VAR_INPUT
    ESS : BOOL;
    TouchSensor01 : BOOL;
    EncoderStartPosition01 : UDINT;
    EncoderStartPosition02 : UDINT;
    TOF_Time_TSR : TIME;
    AutomaticMode : BOOL;
END_VAR

VAR_OUTPUT
    DO_MovingVerticalVSG_01 : BOOL;
END_VAR

VSG_VerticalMoveWithEncoder(
    MethodCall := MethodCall_VerticalMove,
    EmergencyStopSignal := NOT ESS,
    Direction := DirectionVertical,
    InitStateDrive_Input := FALSE,
    DI01 := TouchSensor01,
    DI02_EncoderStart01 := EncoderStartPosition01,
    DI03_EncoderTarget01 := EncoderTargetPosition01,
    DI04_EncoderStart02 := EncoderStartPosition02,
    DI05_EncoderTarget02 := EncoderTargetPosition02,
    TouchSensorRelief := TSR,
    TOF_Time_MotorControl := T#0MS,
    TOF_Time_TouchSensorRelief := TOF_Time_TSR,
    OperatingMode := AutomaticMode
);

DO_MovingVerticalVSG_01 := VSG_VerticalMoveWithEncoder.DigitalOutputControl_01;
ResetMethodCall := VSG_VerticalMoveWithEncoder.ResetMethodCall;

IF ResetMethodCall THEN
    MethodCall_VerticalMove := FALSE;
    jobRunning := FALSE;
    jobFinished := TRUE;
    state := 100;
END_IF;

{attribute 'TcRpcEnable' := '1'}
METHOD Abort : HRESULT
VAR_INPUT
    hdl : UDINT;
END_VAR
callCounterAbort := callCounterAbort + 1;

MethodCall_VerticalMove := FALSE;
DO_MovingVerticalVSG_01 := FALSE;

jobRunning := FALSE;
jobFinished := TRUE;
state := 999;

Abort := 0;
END_METHOD

{attribute 'TcRpcEnable' := '1'}
METHOD CheckState : HRESULT
VAR_INPUT
    hdl : UDINT;
END_VAR

VAR_OUTPUT
    bBusy : BOOL;
    State : UDINT;
    IsDone : BOOL;
END_VAR
callCounterCheckState := callCounterCheckState + 1;

bBusy := jobRunning;
State := state;
IsDone := jobFinished;

CheckState := 0;
END_METHOD

{attribute 'TcRpcEnable' := '1'}
METHOD Start : HRESULT
VAR_INPUT
    MethodCall : BOOL;
    MovementDirection : BOOL;
    EncoderPositionVertical_01 : UDINT;
    EncoderPositionVertical_02 : UDINT;
    TouchSensorRelief : BOOL;
END_VAR

VAR_OUTPUT
    hdl : UDINT;
END_VAR
callCounterStart := callCounterStart + 1;

IF NOT jobRunning THEN

    MethodCall_VerticalMove := MethodCall;
    DirectionVertical := MovementDirection;

    EncoderTargetPosition01 := EncoderPositionVertical_01;
    EncoderTargetPosition02 := EncoderPositionVertical_02;

    TSR := TouchSensorRelief;

    jobRunning := TRUE;
    jobFinished := FALSE;
    state := 1;

    hdl := 1;
    Start := 0;

ELSE

    hdl := 0;
    Start := 16#800700AA;

END_IF;
END_METHOD

END_FUNCTION_BLOCK

// ---- POUs/Moduls/VSG_Skills/VSG_AS_RotationMoveEncoder.TcPOU
{attribute 'OPC.UA.DA.JobMethod' := 'JobMethode_RotationMove'}
FUNCTION_BLOCK VSG_AS_RotationMoveEncoder
VAR
    MethodCall_RotationMove : BOOL := FALSE;
    ResetMethodCall : BOOL := FALSE;

    DirectionRotation : BOOL := TRUE;

    EncoderTargetPosition01 : UDINT;
    EncoderTargetPosition02 : UDINT;

    TSR : BOOL := FALSE;

    callCounterStart : ULINT;
    callCounterCheckState : ULINT;
    callCounterAbort : ULINT;

    jobRunning : BOOL := FALSE;
    jobFinished : BOOL := FALSE;
    state : UDINT := 0;

    VSG_RotationMoveWithEncoder : AxisControl_Encoder;
END_VAR

VAR_INPUT
    ESS : BOOL;
    TouchSensor01 : BOOL;
    EncoderStartPosition01 : UDINT;
    EncoderStartPosition02 : UDINT;
    TOF_Time_TSR : TIME;
    AutomaticMode : BOOL;
END_VAR

VAR_OUTPUT
    DO_MovingRotationVSG_01 : BOOL;
END_VAR

VSG_RotationMoveWithEncoder(
    MethodCall := MethodCall_RotationMove,
    EmergencyStopSignal := NOT ESS,
    Direction := DirectionRotation,
    InitStateDrive_Input := FALSE,
    DI01 := TouchSensor01,
    DI02_EncoderStart01 := EncoderStartPosition01,
    DI03_EncoderTarget01 := EncoderTargetPosition01,
    DI04_EncoderStart02 := EncoderStartPosition02,
    DI05_EncoderTarget02 := EncoderTargetPosition02,
    TouchSensorRelief := TSR,
    TOF_Time_MotorControl := T#0MS,
    TOF_Time_TouchSensorRelief := TOF_Time_TSR,
    OperatingMode := AutomaticMode
);

DO_MovingRotationVSG_01 := VSG_RotationMoveWithEncoder.DigitalOutputControl_01;
ResetMethodCall := VSG_RotationMoveWithEncoder.ResetMethodCall;

IF ResetMethodCall THEN
    MethodCall_RotationMove := FALSE;
    jobRunning := FALSE;
    jobFinished := TRUE;
    state := 100;
END_IF;

{attribute 'TcRpcEnable' := '1'}
METHOD Abort : HRESULT
VAR_INPUT
    hdl : UDINT;
END_VAR
callCounterAbort := callCounterAbort + 1;

MethodCall_RotationMove := FALSE;
DO_MovingRotationVSG_01 := FALSE;

jobRunning := FALSE;
jobFinished := TRUE;
state := 999;

Abort := 0;
END_METHOD

{attribute 'TcRpcEnable' := '1'}
METHOD CheckState : HRESULT
VAR_INPUT
    hdl : UDINT;
END_VAR

VAR_OUTPUT
    bBusy : BOOL;
    State : UDINT;
    IsDone : BOOL;
END_VAR
callCounterCheckState := callCounterCheckState + 1;

bBusy := jobRunning;
State := state;
IsDone := jobFinished;

CheckState := 0;
END_METHOD

{attribute 'TcRpcEnable' := '1'}
METHOD Start : HRESULT
VAR_INPUT
    MethodCall : BOOL;
    MovementDirection : BOOL;
    EncoderPositionRotation_01 : UDINT;
    EncoderPositionRotation_02 : UDINT;
    TouchSensorRelief : BOOL;
END_VAR

VAR_OUTPUT
    hdl : UDINT;
END_VAR
callCounterStart := callCounterStart + 1;

IF NOT jobRunning THEN

    MethodCall_RotationMove := MethodCall;
    DirectionRotation := MovementDirection;

    EncoderTargetPosition01 := EncoderPositionRotation_01;
    EncoderTargetPosition02 := EncoderPositionRotation_02;

    TSR := TouchSensorRelief;

    jobRunning := TRUE;
    jobFinished := FALSE;
    state := 1;

    hdl := 1;
    Start := 0;

ELSE

    hdl := 0;
    Start := 16#800700AA;

END_IF;
END_METHOD

END_FUNCTION_BLOCK

// ---- POUs/Moduls/VSG_Skills/VSG_AS_CompressorControl.TcPOU
{attribute 'OPC.UA.DA.JobMethod' := 'JobMethode_CompressorControl'}
FUNCTION_BLOCK VSG_AS_CompressorControl
VAR
    MethodCall_CompressorControl : BOOL := FALSE;
    ResetMethodCall : BOOL := FALSE;

    Destination : BOOL := TRUE;

    EncoderTargetPosition01 : UDINT;
    EncoderTargetPosition02 : UDINT;
    EncoderTargetPosition03 : UDINT;
    EncoderTargetPosition04 : UDINT;
    EncoderTargetPosition05 : UDINT;
    EncoderTargetPosition06 : UDINT;

    callCounterStart : ULINT;
    callCounterCheckState : ULINT;
    callCounterAbort : ULINT;

    jobRunning : BOOL := FALSE;
    jobFinished : BOOL := FALSE;
    state : UDINT := 0;

    MBS_VSG_VerticalMove : CompressorControl;

    TON_TimeCompressor : TIME := T#0MS;
    TON_TimeValve : TIME := T#0MS;
    TON_TimePowerOffSelfSet : TIME := T#100MS;

    PowerOffSelfSet : BOOL := TRUE;
END_VAR

VAR_INPUT
    ESS : BOOL;

    EncoderStartPosition01 : UDINT;
    EncoderStartPosition02 : UDINT;
    EncoderStartPosition03 : UDINT;
    EncoderStartPosition04 : UDINT;
    EncoderStartPosition05 : UDINT;
    EncoderStartPosition06 : UDINT;

    WorkpieceAtPickupPosition : BOOL;
    AutomaticMode : BOOL;
END_VAR

VAR_OUTPUT
    DO_CompressorVSG : BOOL;
    DO_ValveVSG : BOOL;

    VSG_ErrorDetected : BOOL;
    VSG_ErrorCode : UDINT;
END_VAR

//VSG_ErrorDetected := FALSE;
//VSG_ErrorCode := 0;

IF MethodCall_CompressorControl AND NOT WorkpieceAtPickupPosition THEN

    VSG_ErrorDetected := TRUE;
    VSG_ErrorCode := 1001;

    DO_CompressorVSG := FALSE;
    DO_ValveVSG := FALSE;

    MethodCall_CompressorControl := FALSE;
    ResetMethodCall := TRUE;

    jobRunning := FALSE;
    jobFinished := TRUE;
    state := 900;

ELSE

    MBS_VSG_VerticalMove(
        MethodCall := MethodCall_CompressorControl,
        EmergencyStopSignal := NOT ESS,
        Destination := Destination,
        InitStateDrive_Input := FALSE,

        DI01 := WorkpieceAtPickupPosition,
        DI02 := FALSE,

        DI03_EncoderStart01 := EncoderStartPosition01,
        DI04_EncoderStart02 := EncoderStartPosition02,
        DI05_EncoderStart03 := EncoderStartPosition03,
        DI06_EncoderStart04 := EncoderStartPosition04,
        DI07_EncoderStart05 := EncoderStartPosition05,
        DI08_EncoderStart06 := EncoderStartPosition06,

        DI09_EncoderTarget01 := EncoderTargetPosition01,
        DI10_EncoderTarget02 := EncoderTargetPosition02,
        DI11_EncoderTarget03 := EncoderTargetPosition03,
        DI12_EncoderTarget04 := EncoderTargetPosition04,
        DI13_EncoderTarget05 := EncoderTargetPosition05,
        DI14_EncoderTarget06 := EncoderTargetPosition06,

        PowerOFF_SelfSet := PowerOffSelfSet,
        TON_Time_PowerOFFSelfSet := TON_TimePowerOffSelfSet,
        TON_Time_Compressor := TON_TimeCompressor,
        TON_Time_Valve := TON_TimeValve,
        OperatingMode := AutomaticMode
    );

    DO_CompressorVSG := MBS_VSG_VerticalMove.DigitalOutputControl_01;
    DO_ValveVSG := MBS_VSG_VerticalMove.DigitalOutputControl_02;
    ResetMethodCall := MBS_VSG_VerticalMove.ResetMethodCall;

    IF ResetMethodCall THEN
        MethodCall_CompressorControl := FALSE;
        jobRunning := FALSE;
        jobFinished := TRUE;
        state := 100;
    END_IF;

END_IF;

{attribute 'TcRpcEnable' := '1'}
METHOD Abort : HRESULT
VAR_INPUT
    hdl : UDINT;
END_VAR
callCounterAbort := callCounterAbort + 1;

MethodCall_CompressorControl := FALSE;
ResetMethodCall := TRUE;

DO_CompressorVSG := FALSE;
DO_ValveVSG := FALSE;

jobRunning := FALSE;
jobFinished := TRUE;
state := 999;

Abort := 0;
END_METHOD

{attribute 'TcRpcEnable' := '1'}
METHOD CheckState : HRESULT
VAR_INPUT
    hdl : UDINT;
END_VAR

VAR_OUTPUT
    bBusy : BOOL;
    State : UDINT;
    IsDone : BOOL;
    HasError : BOOL;
    ErrorCode : UDINT;
END_VAR
callCounterCheckState := callCounterCheckState + 1;

bBusy := jobRunning;
State := state;
IsDone := jobFinished;
HasError := VSG_ErrorDetected;
ErrorCode := VSG_ErrorCode;

CheckState := 0;
END_METHOD

{attribute 'TcRpcEnable' := '1'}
METHOD Start : HRESULT
VAR_INPUT
    MethodCall : BOOL;
    DestinationReached : BOOL;
    EncoderTargetPosition_01 : UDINT;
    EncoderTargetPosition_02 : UDINT;
    EncoderTargetPosition_03 : UDINT;
    EncoderTargetPosition_04 : UDINT;
    EncoderTargetPosition_05 : UDINT;
    EncoderTargetPosition_06 : UDINT;
END_VAR

VAR_OUTPUT
    hdl : UDINT;
END_VAR
callCounterStart := callCounterStart + 1;

IF NOT jobRunning THEN
	
	IF MethodCall THEN
        OPCUA.lastExecutedProcess := 'VSG_Skill_SuctionProcess';
        OPCUA.lastExecutedSkill := 'VSG_AS_CompressorControl';
    END_IF;
	
    MethodCall_CompressorControl := MethodCall;
    Destination := DestinationReached;

    EncoderTargetPosition01 := EncoderTargetPosition_01;
    EncoderTargetPosition02 := EncoderTargetPosition_02;
    EncoderTargetPosition03 := EncoderTargetPosition_03;
    EncoderTargetPosition04 := EncoderTargetPosition_04;
    EncoderTargetPosition05 := EncoderTargetPosition_05;
    EncoderTargetPosition06 := EncoderTargetPosition_06;

    jobRunning := TRUE;
    jobFinished := FALSE;
    state := 1;

    hdl := 1;
    Start := 0;

ELSE

    hdl := 0;
    Start := 16#800700AA;

END_IF;
END_METHOD

END_FUNCTION_BLOCK

// ---- POUs/AtomicSkillsSchablonen/CompressorControl.TcPOU
FUNCTION_BLOCK CompressorControl
VAR_INPUT
    MethodCall : BOOL;
    EmergencyStopSignal : BOOL;
    Destination : BOOL;
    InitStateDrive_Input : BOOL;

    DI01 : BOOL;
    DI02 : BOOL;

    DI03_EncoderStart01 : UDINT;
    DI04_EncoderStart02 : UDINT;
    DI05_EncoderStart03 : UDINT;
    DI06_EncoderStart04 : UDINT;
    DI07_EncoderStart05 : UDINT;
    DI08_EncoderStart06 : UDINT;

    DI09_EncoderTarget01 : UDINT;
    DI10_EncoderTarget02 : UDINT;
    DI11_EncoderTarget03 : UDINT;
    DI12_EncoderTarget04 : UDINT;
    DI13_EncoderTarget05 : UDINT;
    DI14_EncoderTarget06 : UDINT;

    PowerOFF_SelfSet : BOOL;
    TON_Time_PowerOFFSelfSet : TIME;
    TON_Time_Compressor : TIME;
    TON_Time_Valve : TIME;
    OperatingMode : BOOL;
END_VAR

VAR_OUTPUT
    DigitalOutputControl_01 : BOOL;
    DigitalOutputControl_02 : BOOL;
    ResetMethodCall : BOOL;
END_VAR

VAR
    RS_Compressor : RS;
    RS_Valve : RS;

    TON_Compressor_Control : TON;
    TON_Valve_Control : TON;
    TON_SelfSet : TON;

    R_TRIG_MethodCall : R_TRIG;

    R_TRIG_EncoderPos01_CompressorInput : R_TRIG;
    R_TRIG_EncoderPos02_CompressorInput : R_TRIG;
    R_TRIG_EncoderPos03_CompressorInput : R_TRIG;
    R_TRIG_EncoderPos04_CompressorInput : R_TRIG;
    R_TRIG_EncoderPos05_CompressorInput : R_TRIG;
    R_TRIG_EncoderPos06_CompressorInput : R_TRIG;

    R_TRIG_EncoderPos01_CompressorOutput : R_TRIG;
    R_TRIG_EncoderPos02_CompressorOutput : R_TRIG;
    R_TRIG_EncoderPos03_CompressorOutput : R_TRIG;
    R_TRIG_EncoderPos04_CompressorOutput : R_TRIG;
    R_TRIG_EncoderPos05_CompressorOutput : R_TRIG;
    R_TRIG_EncoderPos06_CompressorOutput : R_TRIG;

    R_TRIG_EncoderPos01_ValveInput : R_TRIG;
    R_TRIG_EncoderPos02_ValveInput : R_TRIG;
    R_TRIG_EncoderPos03_ValveInput : R_TRIG;
    R_TRIG_EncoderPos04_ValveInput : R_TRIG;
    R_TRIG_EncoderPos05_ValveInput : R_TRIG;
    R_TRIG_EncoderPos06_ValveInput : R_TRIG;

    R_TRIG_EncoderPos01_ValveOutput : R_TRIG;
    R_TRIG_EncoderPos02_ValveOutput : R_TRIG;
    R_TRIG_EncoderPos03_ValveOutput : R_TRIG;
    R_TRIG_EncoderPos04_ValveOutput : R_TRIG;
    R_TRIG_EncoderPos05_ValveOutput : R_TRIG;
    R_TRIG_EncoderPos06_ValveOutput : R_TRIG;

    bEncoderInputCondition : BOOL;
    bEncoderOutputCondition : BOOL;
    bStartCondition : BOOL;
    bResetCondition : BOOL;
END_VAR

R_TRIG_MethodCall(CLK := MethodCall);

R_TRIG_EncoderPos01_CompressorInput(CLK := DI03_EncoderStart01 <> DI09_EncoderTarget01);
R_TRIG_EncoderPos02_CompressorInput(CLK := DI04_EncoderStart02 <> DI10_EncoderTarget02);
R_TRIG_EncoderPos03_CompressorInput(CLK := DI05_EncoderStart03 <> DI11_EncoderTarget03);
R_TRIG_EncoderPos04_CompressorInput(CLK := DI06_EncoderStart04 <> DI12_EncoderTarget04);
R_TRIG_EncoderPos05_CompressorInput(CLK := DI07_EncoderStart05 <> DI13_EncoderTarget05);
R_TRIG_EncoderPos06_CompressorInput(CLK := DI08_EncoderStart06 <> DI14_EncoderTarget06);

R_TRIG_EncoderPos01_CompressorOutput(CLK := DI03_EncoderStart01 = DI09_EncoderTarget01);
R_TRIG_EncoderPos02_CompressorOutput(CLK := DI04_EncoderStart02 = DI10_EncoderTarget02);
R_TRIG_EncoderPos03_CompressorOutput(CLK := DI05_EncoderStart03 = DI11_EncoderTarget03);
R_TRIG_EncoderPos04_CompressorOutput(CLK := DI06_EncoderStart04 = DI12_EncoderTarget04);
R_TRIG_EncoderPos05_CompressorOutput(CLK := DI07_EncoderStart05 = DI13_EncoderTarget05);
R_TRIG_EncoderPos06_CompressorOutput(CLK := DI08_EncoderStart06 = DI14_EncoderTarget06);

R_TRIG_EncoderPos01_ValveInput(CLK := DI03_EncoderStart01 <> DI09_EncoderTarget01);
R_TRIG_EncoderPos02_ValveInput(CLK := DI04_EncoderStart02 <> DI10_EncoderTarget02);
R_TRIG_EncoderPos03_ValveInput(CLK := DI05_EncoderStart03 <> DI11_EncoderTarget03);
R_TRIG_EncoderPos04_ValveInput(CLK := DI06_EncoderStart04 <> DI12_EncoderTarget04);
R_TRIG_EncoderPos05_ValveInput(CLK := DI07_EncoderStart05 <> DI13_EncoderTarget05);
R_TRIG_EncoderPos06_ValveInput(CLK := DI08_EncoderStart06 <> DI14_EncoderTarget06);

R_TRIG_EncoderPos01_ValveOutput(CLK := DI03_EncoderStart01 = DI09_EncoderTarget01);
R_TRIG_EncoderPos02_ValveOutput(CLK := DI04_EncoderStart02 = DI10_EncoderTarget02);
R_TRIG_EncoderPos03_ValveOutput(CLK := DI05_EncoderStart03 = DI11_EncoderTarget03);
R_TRIG_EncoderPos04_ValveOutput(CLK := DI06_EncoderStart04 = DI12_EncoderTarget04);
R_TRIG_EncoderPos05_ValveOutput(CLK := DI07_EncoderStart05 = DI13_EncoderTarget05);
R_TRIG_EncoderPos06_ValveOutput(CLK := DI08_EncoderStart06 = DI14_EncoderTarget06);

bEncoderInputCondition :=
    R_TRIG_EncoderPos01_CompressorInput.Q
    AND R_TRIG_EncoderPos02_CompressorInput.Q
    AND R_TRIG_EncoderPos03_CompressorInput.Q
    AND R_TRIG_EncoderPos04_CompressorInput.Q
    AND R_TRIG_EncoderPos05_CompressorInput.Q
    AND R_TRIG_EncoderPos06_CompressorInput.Q;

bEncoderOutputCondition :=
    R_TRIG_EncoderPos01_CompressorOutput.Q
    AND R_TRIG_EncoderPos02_CompressorOutput.Q
    AND R_TRIG_EncoderPos03_CompressorOutput.Q
    AND R_TRIG_EncoderPos04_CompressorOutput.Q
    AND R_TRIG_EncoderPos05_CompressorOutput.Q
    AND R_TRIG_EncoderPos06_CompressorOutput.Q;

bStartCondition :=
    (DI01 OR bEncoderInputCondition OR InitStateDrive_Input)
    AND OperatingMode;

bResetCondition :=
    (Destination AND (DI02 OR bEncoderOutputCondition))
    OR EmergencyStopSignal;

ResetMethodCall := bResetCondition;

RS_Compressor(
    SET := R_TRIG_MethodCall.Q AND bStartCondition,
    RESET1 := bResetCondition
);

TON_Compressor_Control(
    IN := RS_Compressor.Q1,
    PT := TON_Time_Compressor
);

DigitalOutputControl_01 := TON_Compressor_Control.Q;

TON_SelfSet(
    IN := R_TRIG_MethodCall.Q AND PowerOFF_SelfSet,
    PT := TON_Time_PowerOFFSelfSet
);

RS_Valve(
    SET := R_TRIG_MethodCall.Q AND (DI01 OR bEncoderInputCondition OR InitStateDrive_Input),
    RESET1 := (Destination AND (DI02 OR bEncoderOutputCondition OR TON_SelfSet.Q)) OR EmergencyStopSignal
);

TON_Valve_Control(
    IN := RS_Valve.Q1,
    PT := TON_Time_Valve
);

DigitalOutputControl_02 := TON_Valve_Control.Q;

END_FUNCTION_BLOCK

// ---- POUs/ControlOfOutputs/VSG_ControlOfOutputs.TcPOU
FUNCTION_BLOCK VSG_ControlOfOutputs
VAR_INPUT
	F4							: BOOL;
	F1							: BOOL;
	A2							: BOOL;
	A1							: BOOL;
	A6							: BOOL;
	Start						: BOOL;
	VSG_VertikalDown01			: BOOL; 
	VSG_VertikalDown02			: BOOL; 
	VSG_VertikalUp01			: BOOL;
	VSG_VertikalUp02			: BOOL; 
	VSG_HorizontalForwards01 	: BOOL; 
	VSG_HorizontalForwards02	: BOOL;
	VSG_HorizontalBackwards01 	: BOOL; 
	VSG_HorizontalBackwards02 	: BOOL;
	VSG_RotationCW01		 	: BOOL; 
	VSG_RotationCW02		 	: BOOL;
	VSG_RotationCCW01		 	: BOOL; 
	VSG_RotationCCW02		 	: BOOL;
	VSG_Compressor				: BOOL;
	VSG_Valve					: BOOL;
	Init_VSG_VertikalUp			: BOOL;
	Init_VSG_VertikalDown		: BOOL;	
	Init_VSG_HorizontalForwards : BOOL;
	Init_VSG_HorizontalBackwards: BOOL;
	Init_VSG_RotationCW			: BOOL;
	Init_VSG_RotationCCW		: BOOL;

END_VAR
VAR_OUTPUT
	MoveVerticalDown : BOOL;
	MoveVerticalUp : BOOL;
	MoveHorizontalForwards : BOOL;
	MoveHorizontalBackwards : BOOL;
	MoveRotationCW	: BOOL;
	MoveRotationCCW : BOOL;
	CompressorON : BOOL;
	ValveON : BOOL;
	Light_Q1: BOOL;
	Light_Q2: BOOL;
	Light_Q3: BOOL;
END_VAR
VAR
END_VAR

MoveVerticalDown := ((((((F1) OR (A2))) AND (((VSG_VertikalDown01) OR (VSG_VertikalDown02) OR (Init_VSG_VertikalDown))))) OR (((Start) AND (F4))));
MoveVerticalUp := ((((((F1) OR (A2))) AND (((VSG_VertikalUp01) OR (VSG_VertikalUp02) OR (Init_VSG_VertikalUp))))) OR (((Start) AND (F4))));
MoveHorizontalForwards := ((((((F1) OR (A2))) AND (((VSG_HorizontalForwards01) OR (VSG_HorizontalForwards02) OR (Init_VSG_HorizontalForwards))))) OR (((Start) AND (F4))));
MoveHorizontalBackwards := ((((((F1) OR (A2))) AND (((VSG_HorizontalBackwards01) OR (VSG_HorizontalBackwards02) OR (Init_VSG_HorizontalBackwards))))) OR (((Start) AND (F4))));
MoveRotationCW := ((((((F1) OR (A2))) AND (((VSG_RotationCW01) OR (VSG_RotationCW02) OR (Init_VSG_RotationCW))))) OR (((Start) AND (F4))));
MoveRotationCCW := ((((((F1) OR (A2))) AND (((VSG_RotationCCW01) OR (VSG_RotationCCW02) OR (Init_VSG_RotationCCW))))) OR (((Start) AND (F4))));
CompressorON := ((((((F1) OR (A2))) AND (VSG_Compressor))) OR (((Start) AND (F4))));
ValveON := ((((((F1) OR (A2))) AND (VSG_Valve))) OR (((Start) AND (F4))));
Light_Q1 := F1;
Light_Q2 := F4;
Light_Q3 := A1;

END_FUNCTION_BLOCK

// ---- POUs/OperatingModes/VSG_OperatingModes.TcPOU
FUNCTION_BLOCK VSG_OperatingModes
VAR_INPUT
	Start 			: BOOL;
	Stop			: BOOL;
	Reset			: BOOL;
	Schalter		: BOOL;
	Schrittkette_GS	: BOOL;
	Count1 : INT := 0;
	Count2 : INT := 0;
	Alt_abort: BOOL;
	Err_detected: BOOL;
	Diag_finished: BOOL;
	Alt_found: BOOL;
	Cycle_finished: BOOL;

END_VAR
VAR_OUTPUT
	{attribute 'OPC.UA.DA' := '1'} // für OPC UA freigeben
	A1 : BOOL := FALSE; //Initialzustand
	{attribute 'OPC.UA.DA' := '1'} // für OPC UA freigeben
	A2 : BOOL; //Stillstand angefordert am Ende des Zyklus
//	A3 : BOOL; //Stillstand angefordert in einem bestimmten Zustand
//	A4 : BOOL; //Erhaltener Stillstand
	{attribute 'OPC.UA.DA' := '1'} // für OPC UA freigeben
	A5 : BOOL; //Vorbereitung zur Wiederaufnahme nach Störung
	{attribute 'OPC.UA.DA' := '1'} // für OPC UA freigeben
	A6 : BOOL; //Fahrt in den Initialzustand
	{attribute 'OPC.UA.DA' := '1'} // für OPC UA freigeben
	F1 : BOOL; //Normalbetrieb
//	F2 : BOOL; //Anfahren
//	F3 : BOOL; //Abfahren
	{attribute 'OPC.UA.DA' := '1'} // für OPC UA freigeben
	F4 : BOOL; //Handbetrieb
//	F5 : BOOL; //Schrittbetrieb
//	F6 : BOOL; //Testbetrieb
{attribute 'OPC.UA.DA' := '1'} // für OPC UA freigeben
	D1 : BOOL; //Not-Aus
	{attribute 'OPC.UA.DA' := '1'} // für OPC UA freigeben
	D2 : BOOL; //Diagnose und Störbehandlung
	{attribute 'OPC.UA.DA' := '1'} // für OPC UA freigeben
	D3 : BOOL; //Produktion trotz Störung
	MethodCall_InitStateDrive : BOOL;
	InputVar_InitStateDrive : BOOL;
END_VAR
VAR
	bFirstScan : BOOL := TRUE;
	FirstScanCount: INT := 0;
	AlwaysTrue : BOOL := TRUE;
	TestingVariable : BOOL;	
	 nTaskIdx : DINT;
	RS_InitialState: RS;
	RS_InitialState11: RS;	
	RS_InitialDrive: RS;
	RS_ManualOperationMode: RS;
	RS_AutomaticOperationMode: RS;
	RS_CycleEnded: RS;
	//Count: INT := 0;
	R_TRIG_Manual: R_TRIG;
	R_TRIG_Automatic: R_TRIG;
	R_TRIG_InitialDrive: R_TRIG;
	R_TRIG_CycleEnded: R_TRIG;
	R_TRIG_Init: R_TRIG;
	NeverTrue: BOOL := FALSE;
	SR_D1: SR;
	RS_D2: RS;
	
	RS_D3: RS;
	RS_A5: RS;
	
	
	bFirstCycle: BOOL;
END_VAR
VAR // added by the converter: edge detectors and wires of the graphical bodies
    _w1, _w2, _w3, _w4 : BOOL;
END_VAR

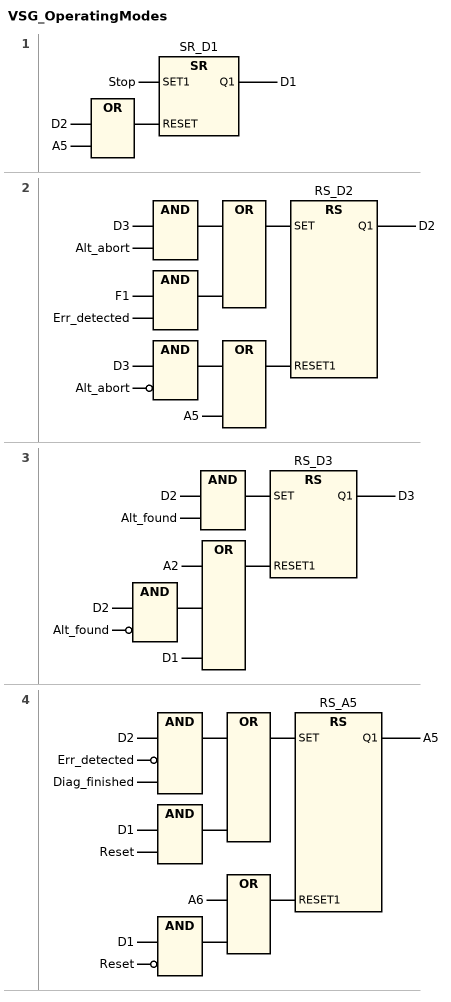
// NETWORK 1
SR_D1(SET1 := Stop, RESET := D2 OR A5); // SR
D1 := SR_D1.Q1;

// NETWORK 2
RS_D2(SET := D3 AND Alt_abort OR F1 AND Err_detected, RESET1 := D3 AND NOT Alt_abort OR A5); // RS
D2 := RS_D2.Q1;

// NETWORK 3
RS_D3(SET := D2 AND Alt_found, RESET1 := A2 OR D2 AND NOT Alt_found OR D1); // RS
D3 := RS_D3.Q1;

// NETWORK 4
RS_A5(SET := D2 AND NOT Err_detected AND Diag_finished OR D1 AND Reset, RESET1 := A6 OR D1 AND NOT Reset); // RS
A5 := RS_A5.Q1;

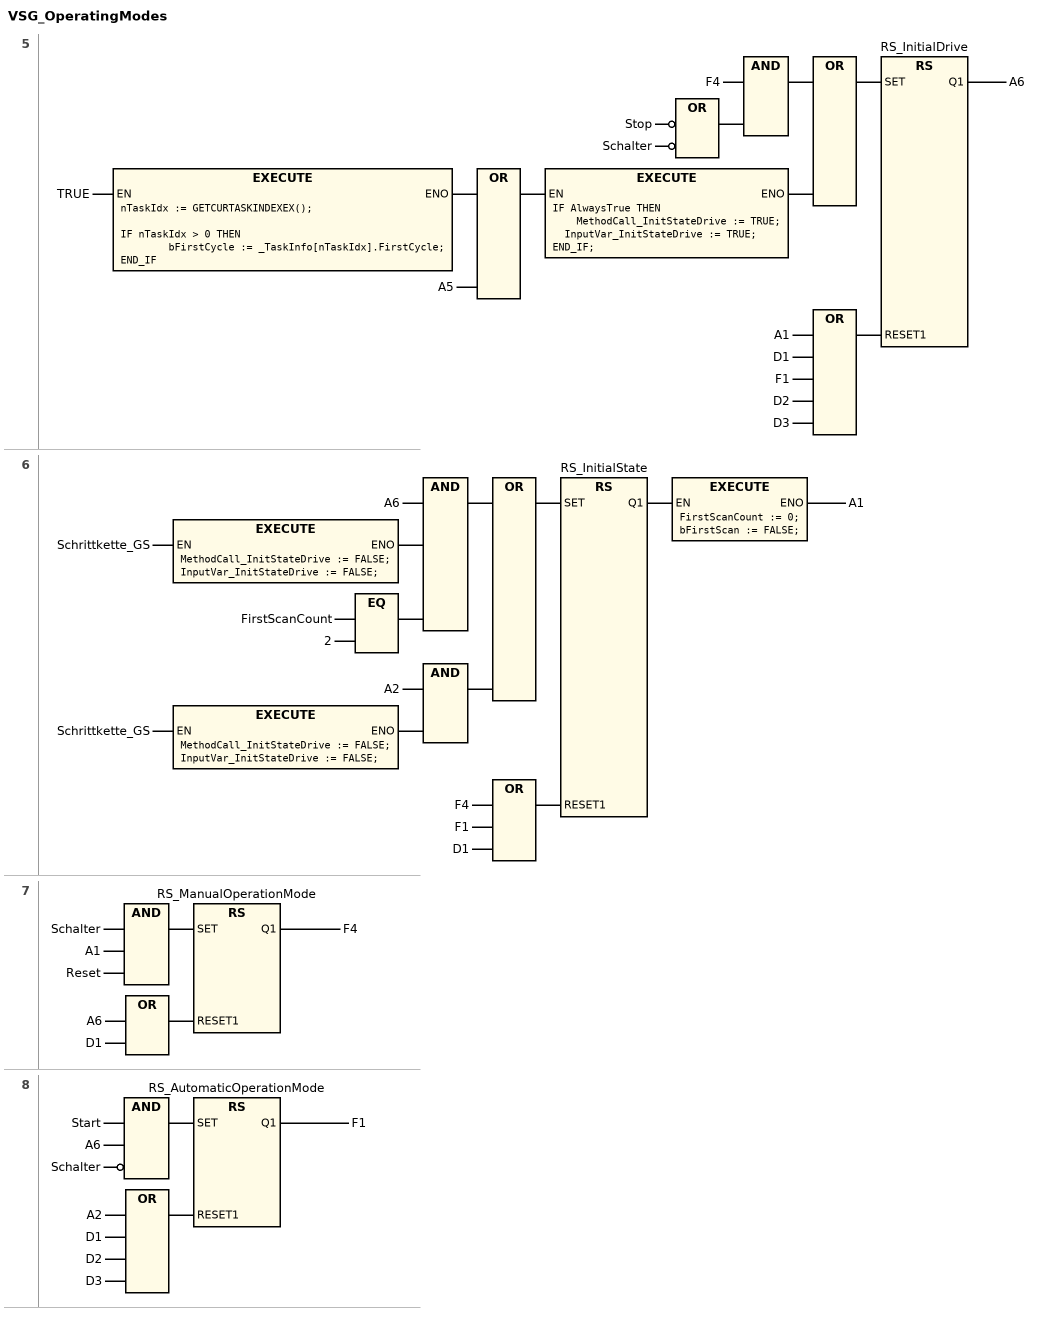
// NETWORK 5
nTaskIdx := GETCURTASKINDEXEX();

IF nTaskIdx > 0 THEN
        bFirstCycle := _TaskInfo[nTaskIdx].FirstCycle;
END_IF
_w1 := TRUE OR A5;
IF _w1 THEN
    IF AlwaysTrue THEN
        MethodCall_InitStateDrive := TRUE;
    	InputVar_InitStateDrive := TRUE;
    END_IF;
END_IF
RS_InitialDrive(SET := F4 AND (NOT Stop OR NOT Schalter) OR _w1, RESET1 := A1 OR D1 OR F1 OR D2 OR D3); // RS
A6 := RS_InitialDrive.Q1;

// NETWORK 6
_w2 := Schrittkette_GS;
IF _w2 THEN
    MethodCall_InitStateDrive := FALSE;
    InputVar_InitStateDrive := FALSE;
END_IF
_w3 := Schrittkette_GS;
IF _w3 THEN
    MethodCall_InitStateDrive := FALSE;
    InputVar_InitStateDrive := FALSE;
END_IF
RS_InitialState(SET := A6 AND _w2 AND FirstScanCount = 2 OR A2 AND _w3, RESET1 := F4 OR F1 OR D1); // RS
_w4 := RS_InitialState.Q1;
IF _w4 THEN
    FirstScanCount := 0;
    bFirstScan := FALSE;
END_IF
A1 := _w4;

// NETWORK 7
RS_ManualOperationMode(SET := Schalter AND A1 AND Reset, RESET1 := A6 OR D1); // RS
F4 := RS_ManualOperationMode.Q1;

// NETWORK 8
RS_AutomaticOperationMode(SET := Start AND A6 AND NOT Schalter, RESET1 := A2 OR D1 OR D2 OR D3); // RS
F1 := RS_AutomaticOperationMode.Q1;

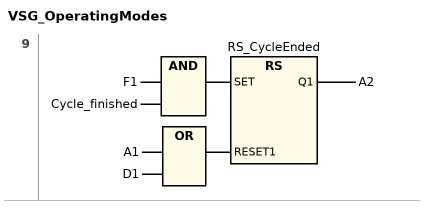
// NETWORK 9
RS_CycleEnded(SET := F1 AND Cycle_finished, RESET1 := A1 OR D1); // RS
A2 := RS_CycleEnded.Q1;

END_FUNCTION_BLOCK

// ---- POUs/DiagnosisHandler/VSG_DiagnosisHandler.TcPOU
FUNCTION_BLOCK VSG_DiagnosisHandler
VAR_INPUT
    Diagnose_gefordert : BOOL;
    ErrorDetectedRaw   : BOOL;
    Reset              : BOOL;
    PulseTime          : TIME := T#100MS;
END_VAR
VAR_OUTPUT
    Err_detected  : BOOL := FALSE;
    Diag_finished : BOOL := FALSE;
    Alt_found     : BOOL := FALSE;
    Busy          : BOOL := FALSE;
END_VAR
VAR
    rtReq      : R_TRIG;
    rtError    : R_TRIG;
    rtDiagAck  : R_TRIG;
    rtAltFound : R_TRIG;
    tpPulse    : TP;
END_VAR

rtReq(CLK := Diagnose_gefordert);
rtError(CLK := ErrorDetectedRaw);
rtDiagAck(CLK := OPCUA.Diag_finished);
rtAltFound(CLK := OPCUA.Alt_found);

IF Reset THEN
    Err_detected := FALSE;
    Diag_finished := FALSE;
    Alt_found := FALSE;
    Busy := FALSE;
    OPCUA.TriggerD2 := FALSE;
END_IF

IF rtError.Q THEN
    Err_detected := TRUE;
    Diag_finished := FALSE;
    Alt_found := FALSE;
	OPCUA.TriggerD2 := TRUE;
END_IF

IF rtReq.Q AND Err_detected AND NOT Busy THEN
    Busy := TRUE;
END_IF

IF OPCUA.TriggerD2 AND Diag_finished THEN
    OPCUA.TriggerD2 := FALSE;
END_IF

IF Busy AND rtDiagAck.Q THEN
    Diag_finished := TRUE;
    Alt_found := FALSE;
    Busy := FALSE;
    OPCUA.Diag_finished := FALSE;
    OPCUA.TriggerD2 := FALSE;
END_IF

IF Busy AND rtAltFound.Q THEN
    Alt_found := TRUE;
    Diag_finished := TRUE;
    Busy := FALSE;
    OPCUA.Alt_found := FALSE;
    OPCUA.TriggerD2 := FALSE;
END_IF

IF NOT Diagnose_gefordert AND (Diag_finished OR Alt_found) THEN
    Err_detected := FALSE;
    Diag_finished := FALSE;
    Alt_found := FALSE;
END_IF

END_FUNCTION_BLOCK

// ---- POUs/InitStateDrive/VSG_InitialStateDrive.TcPOU
FUNCTION_BLOCK VSG_InitialStateDrive
VAR_INPUT
    MethodCall_InitDrive : BOOL;
    ESS : BOOL;
    InputInitDriveMode : BOOL;

    TouchSensor01_Rotation : BOOL;
    TouchSensor02_Vertical : BOOL;
    TouchSensor03_horizontal : BOOL;

    TOF_Time_TSR : TIME;
    InitDriveMode : BOOL;
END_VAR

VAR_OUTPUT
    VSG_Init_RotateCW : BOOL;
    VSG_Init_RotateCCW : BOOL;

    VSG_Init_VerticalUp : BOOL;
    VSG_Init_VerticalDown : BOOL;

    VSG_Init_HorizontalForwards : BOOL;
    VSG_Init_HorizontalBackwards : BOOL;

    ResetMethodCall_RotateCW : BOOL;
    ResetMethodCall_RGB_Vertical : BOOL;
    ResetMethodCall_RGB_Horizontal : BOOL;
END_VAR

VAR
    TSR : BOOL := TRUE;

    DirectionVertical : BOOL := TRUE;
    DirectionHorizontal : BOOL := TRUE;
    DirectionRotation : BOOL := TRUE;

    VSG_InitDrive_Rotate_CW : AxisControl_MultipleInputSensors;
    VSG_InitDrive_Vertical_Up : AxisControl_MultipleInputSensors;
    VSG_InitDrive_Horizontal_Backwards : AxisControl_MultipleInputSensors;
END_VAR

VSG_InitDrive_Rotate_CW(
    MethodCall := MethodCall_InitDrive,
    EmergencyStopSignal := NOT ESS,
    Direction := DirectionRotation,
    InitStateDrive_Input := InputInitDriveMode,
    DI01 := FALSE,
    DI02 := TouchSensor01_Rotation,
    TouchSensorRelief := TSR,
    TOF_Time_MotorControl := T#0MS,
    TOF_Time_TouchSensorRelief := TOF_Time_TSR,
    OperatingMode := InitDriveMode
);

VSG_Init_RotateCW := VSG_InitDrive_Rotate_CW.DigitalOutputControl_01;
VSG_Init_RotateCCW := FALSE;
ResetMethodCall_RotateCW := VSG_InitDrive_Rotate_CW.ResetMethodCall;


VSG_InitDrive_Vertical_Up(
    MethodCall := MethodCall_InitDrive,
    EmergencyStopSignal := NOT ESS,
    Direction := DirectionVertical,
    InitStateDrive_Input := InputInitDriveMode,
    DI01 := FALSE,
    DI02 := TouchSensor02_Vertical,
    TouchSensorRelief := TSR,
    TOF_Time_MotorControl := T#0MS,
    TOF_Time_TouchSensorRelief := TOF_Time_TSR,
    OperatingMode := InitDriveMode
);

VSG_Init_VerticalUp := VSG_InitDrive_Vertical_Up.DigitalOutputControl_01;
VSG_Init_VerticalDown := FALSE;
ResetMethodCall_RGB_Vertical := VSG_InitDrive_Vertical_Up.ResetMethodCall;


VSG_InitDrive_Horizontal_Backwards(
    MethodCall := MethodCall_InitDrive,
    EmergencyStopSignal := NOT ESS,
    Direction := DirectionHorizontal,
    InitStateDrive_Input := InputInitDriveMode,
    DI01 := FALSE,
    DI02 := TouchSensor03_horizontal,
    TouchSensorRelief := TSR,
    TOF_Time_MotorControl := T#0MS,
    TOF_Time_TouchSensorRelief := TOF_Time_TSR,
    OperatingMode := InitDriveMode
);

VSG_Init_HorizontalForwards := FALSE;
VSG_Init_HorizontalBackwards := VSG_InitDrive_Horizontal_Backwards.DigitalOutputControl_01;
ResetMethodCall_RGB_Horizontal := VSG_InitDrive_Horizontal_Backwards.ResetMethodCall;

END_FUNCTION_BLOCK

// ---- POUs/AtomicSkillsSchablonen/AutomaticColorDetection_nichtfertig.TcPOU
FUNCTION_BLOCK AutomaticColorDetection_nichtfertig
VAR_INPUT
	MethodCall : BOOL;
	EmergencyStopSignal : BOOL;
	ColorSensor: INT;
	ColorCode_1: INT;
	ColorCode_2: INT;
	ColorCode_3: INT;
	OperatingMode : BOOL;
END_VAR

VAR_OUTPUT
	Color_1: BOOL;
	Color_2: BOOL;
	Color_3: BOOL;
END_VAR

VAR
END_VAR

Color_1 := ((ColorSensor) = (ColorCode_1));
Color_2 := ((ColorSensor) = (ColorCode_2));
Color_3 := ((ColorSensor) = (Color_3));

END_FUNCTION_BLOCK

// ---- POUs/AtomicSkillsSchablonen/CuttingProcess.TcPOU
FUNCTION_BLOCK CuttingProcess
VAR_INPUT//Input-Variablen des FBs
	MethodCall			: BOOL; // Variable zum aktiven Aufruf einer OPC UA Methode
	EmergencyStopSignal : BOOL; // Variable für Not-Signal
	InitStateDrive_Input: BOOL; //InputVariable für Initialfahrt
	DI01				: BOOL; // Digitaler Input wie bspw. Lichtsensor oder Kontaktsensor
	TOF_Time_CuttingTime: TIME; // Ausschaltverzögerung für die Rücksetzbedingung um eine Bearbeitungszeit zu simulieren
	OperatingMode		: BOOL; // Variable zur Festlegung des benötigten Betriebszustandes für die Auslösung des FBs
END_VAR

VAR_OUTPUT //Output-Variablen des FBs
	DigitalOutputControl_01	: BOOL; //Digitale Output Ansteuerung des Motor 1
	ResetMethodCall			: BOOL; //Outputvariable für den Reset der OPC UA Methode
END_VAR

VAR //Interne-Variablen des FBs
//FlipFlop
	RS_CuttingProcess: RS; //FlipFlop für die Ansteuerung der Schneidemaschine
//Zeitverzögerung
	TOF_CuttingTime: TOF; //Ausschaltverzögerung simulativ für die Bearbeitungszeit
//Flanke	
	R_TRIG_MethodCall: R_TRIG; //Flankenerkennung für eingehenden MethodenCall
END_VAR

R_TRIG_MethodCall(CLK := MethodCall);
R_TRIG_MethodCall(CLK := MethodCall);
TOF_CuttingTime(IN := R_TRIG_MethodCall.Q, PT := TOF_Time_CuttingTime);
ResetMethodCall := ((TOF_CuttingTime.Q) OR (EmergencyStopSignal));
RS_CuttingProcess(SET := ((R_TRIG_MethodCall.Q) AND (((DI01) OR (InitStateDrive_Input))) AND (OperatingMode)), RESET1 := ((TOF_CuttingTime.Q) OR (EmergencyStopSignal)));
DigitalOutputControl_01 := RS_CuttingProcess.Q1;

END_FUNCTION_BLOCK

// ---- POUs/AtomicSkillsSchablonen/HardeningProcess.TcPOU
FUNCTION_BLOCK HardeningProcess
VAR_INPUT//Input-Variablen des FBs
	MethodCall				: BOOL; // Variable zum aktiven Aufruf einer OPC UA Methode
	EmergencyStopSignal 	: BOOL; // Variable für Not-Signal
	InitStateDrive_Input	: BOOL; //InputVariable für Initialfahrt
	DI01					: BOOL; // Digitaler Input wie bspw. Lichtsensor oder Kontaktsensor
	TOF_Time_HardeningTime	: TIME; // Ausschaltverzögerung für die Rücksetzbedingung um eine Bearbeitungszeit zu simulieren
	OperatingMode			: BOOL; // Variable zur Festlegung des benötigten Betriebszustandes für die Auslösung des FBs
END_VAR

VAR_OUTPUT //Output-Variablen des FBs
	DigitalOutputControl_01	: BOOL; //Digitale Output Ansteuerung des Motor 1
	ResetMethodCall			: BOOL; //Outputvariable für den Reset der OPC UA Methode
END_VAR

VAR //Interne-Variablen des FBs
//FlipFlop
	RS_HardeningProcess: RS; //FlipFlop für die Ansteuerung des Ofens
//Zeitverzögerung
	TOF_HardeningTime: TOF; //Ausschaltverzögerung simulativ für die Bearbeitungszeit
//Flanke	
	R_TRIG_MethodCall: R_TRIG; //Flankenerkennung für eingehenden MethodenCall
END_VAR

R_TRIG_MethodCall(CLK := MethodCall);
R_TRIG_MethodCall(CLK := MethodCall);
TOF_HardeningTime(IN := R_TRIG_MethodCall.Q, PT := TOF_Time_HardeningTime);
ResetMethodCall := ((TOF_HardeningTime.Q) AND (EmergencyStopSignal));
RS_HardeningProcess(SET := ((R_TRIG_MethodCall.Q) AND (((DI01) OR (InitStateDrive_Input))) AND (OperatingMode)), RESET1 := ((TOF_HardeningTime.Q) AND (EmergencyStopSignal)));
DigitalOutputControl_01 := RS_HardeningProcess.Q1;

END_FUNCTION_BLOCK

// ---- POUs/AtomicSkillsSchablonen/SecuringWorkpiece.TcPOU
FUNCTION_BLOCK SecuringWorkpiece
VAR_INPUT//Input-Variablen des FBs
	MethodCall				: BOOL; // Variable zum aktiven Aufruf einer OPC UA Methode
	EmergencyStopSignal 	: BOOL; // Variable für Not-Signal 
	InitStateDrive_Input	: BOOL; //InputVariable für Initialfahrt
	DI01 					: BOOL; // Digitaler Input wie bspw. Lichtsensor oder Kontaktsensor 
	TON_Time_Securing		: TIME;	// Einschaltverzögerung um eine Bearbeitungszeit zu simulieren
	TON_Time_SecuringProcess: TIME; // Einschaltverzögerung um einen Einspannprozess zu simulieren
	OperatingMode			: BOOL; // Variable zur Festlegung des benötigten Betriebszustandes für die Auslösung des FBs
END_VAR

VAR_OUTPUT //Output-Variablen des FBs
	DigitalOutputControl_01	: BOOL; //Digitale Output Ansteuerung des Motor 1
	DigitalOutputControl_02	: BOOL; //Digitale Output Ansteuerung des Motor 2
	ResetMethodCall			: BOOL; //Outputvariable für den Reset der OPC UA Methode
END_VAR

VAR //Interne-Variablen des FBs
//FlipFlop
	RS_SecuringProcessCompressorON	: RS; //FlipFlop für die Ansteuerung des Compressors
	RS_SecuringProcessCompressorOFF	: RS; //FlipFlop für die Ansteuerung des Ventils	
//Zeitverzögerung
	TON_SecuringTime_Compressor	: TON; //Einschaltverzögerung für Einspannzeit
	TON_SecuringTime_Valve		: TON; //Einschaltverzögerung für Einspannzeit
	TON_SecuringProcessingTime	: TON; //Einschaltverzögerung zur Simulation von einer Gesamtbearbeitungszeit
//Flanke	
	R_TRIG_MethodCall: R_TRIG; //Flankenerkennung für eingehenden MethodenCall
END_VAR

R_TRIG_MethodCall(CLK := MethodCall);
R_TRIG_MethodCall(CLK := MethodCall);
TON_SecuringProcessingTime(IN := R_TRIG_MethodCall.Q, PT := TON_Time_SecuringProcess);
RS_SecuringProcessCompressorON(SET := ((R_TRIG_MethodCall.Q) AND (((DI01) OR (InitStateDrive_Input))) AND (OperatingMode)), RESET1 := ((TON_SecuringProcessingTime.Q) OR (EmergencyStopSignal)));
TON_SecuringTime_Compressor(IN := RS_SecuringProcessCompressorON.Q1, PT := TON_Time_Securing);
DigitalOutputControl_01 := TON_SecuringTime_Compressor.Q;
R_TRIG_MethodCall(CLK := MethodCall);
R_TRIG_MethodCall(CLK := MethodCall);
TON_SecuringProcessingTime(IN := R_TRIG_MethodCall.Q, PT := TON_Time_SecuringProcess);
ResetMethodCall := ((TON_SecuringProcessingTime.Q) OR (EmergencyStopSignal));
RS_SecuringProcessCompressorOFF(SET := ((R_TRIG_MethodCall.Q) AND (((DI01) OR (InitStateDrive_Input))) AND (OperatingMode)), RESET1 := ((TON_SecuringProcessingTime.Q) OR (EmergencyStopSignal)));
TON_SecuringTime_Valve(IN := RS_SecuringProcessCompressorOFF.Q1, PT := TON_Time_Securing + T#0.5s);
DigitalOutputControl_02 := TON_SecuringTime_Valve.Q;

END_FUNCTION_BLOCK

// ---- POUs/AtomicSkillsSchablonen/StampingProcess.TcPOU
FUNCTION_BLOCK StampingProcess
VAR_INPUT//Input-Variablen des FBs
	MethodCall				: BOOL; // Variable zum aktiven Aufruf einer OPC UA Methode
	EmergencyStopSignal 	: BOOL; // Variable für Not-Signal
	InitStateDrive_Input	: BOOL; //InputVariable für Initialfahrt
	DI01					: BOOL; // Digitaler Input wie bspw. Lichtsensor oder Kontaktsensor
	TOF_Time_StampingTime	: TIME; // Ausschaltverzögerung für die Rücksetzbedingung um eine Bearbeitungszeit zu simulieren
	OperatingMode			: BOOL; // Variable zur Festlegung des benötigten Betriebszustandes für die Auslösung des FBs
END_VAR

VAR_OUTPUT //Output-Variablen des FBs
	DigitalOutputControl_01	: BOOL; //Digitale Output Ansteuerung des Motor 1
	ResetMethodCall			: BOOL; //Outputvariable für den Reset der OPC UA Methode
END_VAR

VAR //Interne-Variablen des FBs
//FlipFlop
	RS_StampingProcess: RS; //FlipFlop für die Ansteuerung der Stanzmaschine
//Zeitverzögerung
	TOF_StampingTime: TOF; //Ausschaltverzögerung simulativ für die Bearbeitungszeit
//Flanke	
	R_TRIG_MethodCall: R_TRIG; //Flankenerkennung für eingehenden MethodenCall
END_VAR


R_TRIG_MethodCall(CLK := MethodCall);
R_TRIG_MethodCall(CLK := MethodCall);
TOF_StampingTime(IN := R_TRIG_MethodCall.Q, PT := TOF_Time_StampingTime);
ResetMethodCall := ((TOF_StampingTime.Q) AND (EmergencyStopSignal));
RS_StampingProcess(SET := ((R_TRIG_MethodCall.Q) AND (((DI01) OR (InitStateDrive_Input))) AND (OperatingMode)), RESET1 := ((TOF_StampingTime.Q) AND (EmergencyStopSignal)));
DigitalOutputControl_01 := RS_StampingProcess.Q1;

END_FUNCTION_BLOCK

// ---- POUs/ControlOfOutputs/MBS_ControlOfOutputs.TcPOU
FUNCTION_BLOCK MBS_ControlOfOutputs
VAR_INPUT
	F4							: BOOL;
	F1							: BOOL;
	A2							: BOOL;
	A1							: BOOL;
	A6							: BOOL;
	Start						: BOOL;
// Output Control
	CB_Forwards 				: BOOL; 
	DmPD_Compressor				: BOOL;
	DmPD_Valve					: BOOL;
	DmPD_RotateCW_VSGtoMR02		: BOOL;	
	DmPD_RotateCW_VSGtoCB		: BOOL;
	DmPD_RotateCW_MR02toCB		: BOOL;
	DmPD_RotateCCW_CBtoMR02		: BOOL;	
	DmPD_RotateCCW_CBtoVSG		: BOOL;
	DmPD_RotateCCW_MR02toVSG	: BOOL;
	MR01_HardeningProcess		: BOOL;
	MR01_HorizontalForwards		: BOOL;
	MR01_HoritzontalBackwards	: BOOL;
	MR01_Compressor				: BOOL;
	MR01_Valve					: BOOL;
	MR02_CuttingProcess			: BOOL;
	VSG_HorizontalForwards		: BOOL;
	VSG_HorizontalBackwards		: BOOL;
	VSG_Valve_VerticalDown		: BOOL;
	VSG_Valve_SuctionToDmPD		: BOOL;
	VSG_Valve_SuctionToMR01		: BOOL;
	VSG_Compressor_VerticalDown : BOOL;
	VSG_Compressor_SuctionToDmPD: BOOL;
	VSG_Compressor_SuctionToMR01: BOOL;
	
// InitDriveMode Output Control	
	Init_DmPD_RotateCCW				: BOOL;
	Init_DmPD_RotateCW				: BOOL;
	Init_MR01_HorizontalForwards	: BOOL;
	Init_MR01_HorizontalBackwards	: BOOL;
	Init_MR02_CuttingProcess		: BOOL;
	Init_VSG_HorizontalForwards		: BOOL;
	Init_VSG_HorizontalBackwards	: BOOL;
END_VAR
VAR_OUTPUT
	ConveyorBeltForward: BOOL;
	CompressorON: BOOL;
	ValveDmPD_ON: BOOL;
	RotateDmPD_CW: BOOL;
	RotateDmPD_CCW: BOOL;
	HardeningProcess : BOOL;
	WorkpieceTableMoveHorizontalForwards : BOOL;
	WorkpieceTableMoveHorizontalBackwards : BOOL;
	ValveMR01_ON : BOOL;
	CuttingProcess_ON : BOOL;
	MoveVSGHorizontalForwards : BOOL;
	MoveVSGHorizontalBackwards : BOOL;
	ValveVSG_VerticalDown_ON : BOOL;
	ValveVSG_Suction_ON : BOOL;
	Light_Q1: BOOL;
	Light_Q2: BOOL;
	Light_Q3: BOOL;
	
END_VAR
VAR
END_VAR

ConveyorBeltForward := ((((((F1) OR (A2))) AND (CB_Forwards))) OR (((Start) AND (F4))));
CompressorON := ((((((F1) OR (A2))) AND (((DmPD_Compressor) OR (MR01_Compressor) OR (VSG_Compressor_VerticalDown) OR (VSG_Compressor_SuctionToDmPD) OR (VSG_Compressor_SuctionToMR01))))) OR (((Start) AND (F4))));
ValveDmPD_ON := ((((((F1) OR (A2))) AND (DmPD_Valve))) OR (((Start) AND (F4))));
RotateDmPD_CW := ((((((F1) OR (A2))) AND (((DmPD_RotateCW_VSGtoMR02) OR (DmPD_RotateCW_MR02toCB) OR (DmPD_RotateCW_VSGtoCB))))) OR (((Start) AND (F4))) OR (((A6) AND (Init_DmPD_RotateCW))));
RotateDmPD_CCW := ((((((F1) OR (A2))) AND (((DmPD_RotateCCW_CBtoMR02) OR (DmPD_RotateCCW_CBtoVSG) OR (DmPD_RotateCCW_MR02toVSG))))) OR (((Start) AND (F4))) OR (((A6) AND (Init_DmPD_RotateCCW))));
HardeningProcess := ((((((F1) OR (A2))) AND (MR01_HardeningProcess))) OR (((Start) AND (F4))));
WorkpieceTableMoveHorizontalForwards := ((((((F1) OR (A2))) AND (MR01_HorizontalForwards))) OR (((Start) AND (F4))) OR (((A6) AND (Init_MR01_HorizontalForwards))));
WorkpieceTableMoveHorizontalBackwards := ((((((F1) OR (A2))) AND (MR01_HoritzontalBackwards))) OR (((Start) AND (F4))) OR (((A6) AND (Init_MR01_HorizontalBackwards))));
ValveMR01_ON := ((((((F1) OR (A2))) AND (MR01_Valve))) OR (((Start) AND (F4))));
CuttingProcess_ON := ((((((F1) OR (A2))) AND (MR02_CuttingProcess))) OR (((Start) AND (F4))) OR (((A6) AND (Init_MR02_CuttingProcess))));
MoveVSGHorizontalForwards := ((((((F1) OR (A2))) AND (VSG_HorizontalForwards))) OR (((Start) AND (F4))) OR (((A6) AND (Init_VSG_HorizontalForwards))));
MoveVSGHorizontalBackwards := ((((((F1) OR (A2))) AND (VSG_HorizontalBackwards))) OR (((Start) AND (F4))) OR (((A6) AND (Init_VSG_HorizontalBackwards))));
ValveVSG_VerticalDown_ON := ((((((F1) OR (A2))) AND (VSG_Valve_VerticalDown))) OR (((Start) AND (F4))));
ValveVSG_Suction_ON := ((((((F1) OR (A2))) AND (((VSG_Valve_SuctionToDmPD) OR (VSG_Valve_SuctionToMR01))))) OR (((Start) AND (F4))));
Light_Q1 := F1;
Light_Q2 := F4;
Light_Q3 := A1;

END_FUNCTION_BLOCK

// ---- POUs/ControlOfOutputs/SST_ControlOfOutputs.TcPOU
FUNCTION_BLOCK SST_ControlOfOutputs
VAR_INPUT
	F4							: BOOL;
	F1							: BOOL;
	A2							: BOOL;
	A1							: BOOL;
	A6							: BOOL;
	Start						: BOOL;	
//Variablen zur Outputsteuerung aus anderen FBs
	//Output-Variablen der Komponente ConveyorBelt	
	CB_MoveForwardToPD01: BOOL;
	CB_MoveForwardToPD02: BOOL;
	CB_MoveForwardToPD03: BOOL;
	CB_MoveForwardTillEnd: BOOL;
	
	//Output-Variablen der Komponente PushingDevice
	PD01_Compressor : BOOL;
	PD02_Compressor : BOOL;
	PD03_Compressor : BOOL;
	PD01_Valve : BOOL;
	PD02_Valve : BOOL;
	PD03_Valve : BOOL;	
	
	//Output-Variablen für Init-Fahrt
	Init_PD01_Compressor : BOOL;
	Init_PD02_Compressor : BOOL;
	Init_PD03_Compressor : BOOL;
	Init_PD01_Valve : BOOL;
	Init_PD02_Valve : BOOL;
	Init_PD03_Valve : BOOL;

END_VAR
VAR_OUTPUT
	ConveyorBeltForward : BOOL;
	CompressorON : BOOL;
	ValvePD01_ON : BOOL;
	ValvePD02_ON : BOOL;
	ValvePD03_ON : BOOL;
	Light_Q1: BOOL;
	Light_Q2: BOOL;
	Light_Q3: BOOL;
	
END_VAR
VAR
END_VAR

ConveyorBeltForward := ((((((F1) OR (A2))) AND (((CB_MoveForwardToPD01) OR (CB_MoveForwardToPD02) OR (CB_MoveForwardToPD03) OR (CB_MoveForwardTillEnd))))) OR (((Start) AND (F4))));
CompressorON := ((((((F1) OR (A2))) AND (((PD01_Compressor) OR (PD02_Compressor) OR (PD03_Compressor) OR (Init_PD01_Compressor) OR (Init_PD02_Compressor) OR (Init_PD03_Compressor))))) OR (((Start) AND (F4))));
ValvePD01_ON := ((((((F1) OR (A2))) AND (((PD01_Valve) OR (Init_PD01_Valve))))) OR (((Start) AND (F4))));
ValvePD02_ON := ((((((F1) OR (A2))) AND (((PD02_Valve) OR (Init_PD02_Valve))))) OR (((Start) AND (F4))));
ValvePD03_ON := ((((((F1) OR (A2))) AND (((PD03_Valve) OR (Init_PD03_Valve))))) OR (((Start) AND (F4))));
Light_Q1 := F1;
Light_Q2 := F4;
Light_Q3 := A1;

END_FUNCTION_BLOCK

// ---- POUs/InitStateDrive/MBS_DmPD_InitialStateDrive.TcPOU
FUNCTION_BLOCK MBS_DmPD_InitialStateDrive
VAR_INPUT
	MethodCall_InitDrive : BOOL;
	ESS : BOOL;
	InputInitialStateDrive : BOOL;
	DI02_CW : BOOL;
	DI01_CCW : BOOL;
	DI02_CCW : BOOL;	
	InitDriveMode : BOOL;
END_VAR
VAR_OUTPUT
	MotorControl_CW : BOOL;
	MotorControl_CCW : BOOL;
	ResetMethodCallRotateCW : BOOL;
	ResetMethodCallRotateCCW : BOOL;
END_VAR
VAR
	DirectionCW : STRING;
	DirectionCCW : STRING;
	MBS_DmPD_InitDrive_Rotate_CW: AxisControl_MultipleInputSensors;
	MBS_DmPD_InitDrive_Rotate_CCW: AxisControl_MultipleInputSensors;
END_VAR

MBS_DmPD_InitDrive_Rotate_CW(
    MethodCall := MethodCall_InitDrive,
    EmergencyStopSignal := ESS,
    Direction := DirectionCW,
    InitStateDrive_Input := InputInitialStateDrive,
    DI01 := ,
    DI02 := DI02_CW,
    TouchSensorRelief := ,
    TOF_Time_MotorControl := ,
    TOF_Time_TouchSensorRelief := ,
    OperatingMode := InitDriveMode
);
MotorControl_CW := MBS_DmPD_InitDrive_Rotate_CW.DigitalOutputControl_01;
MBS_DmPD_InitDrive_Rotate_CCW(
    MethodCall := MethodCall_InitDrive,
    EmergencyStopSignal := ESS,
    Direction := DirectionCCW,
    InitStateDrive_Input := ,
    DI01 := DI01_CCW,
    DI02 := DI02_CCW,
    TouchSensorRelief := ,
    TOF_Time_MotorControl := ,
    TOF_Time_TouchSensorRelief := ,
    OperatingMode := InitDriveMode
);
MotorControl_CCW := MBS_DmPD_InitDrive_Rotate_CCW.DigitalOutputControl_01;

END_FUNCTION_BLOCK

// ---- POUs/InitStateDrive/MBS_MR01_InitialStateDrive.TcPOU
FUNCTION_BLOCK MBS_MR01_InitialStateDrive
VAR_INPUT
	MethodCall_InitDrive : BOOL;
	ESS : BOOL;
	InputInitStateDrive : BOOL;
	TouchSensor01 : BOOL;
	TouchSensor02 : BOOL;
	InitDriveMode : BOOL;
END_VAR
VAR_OUTPUT
	MotorControlHorizontalForwards : BOOL;
	MotorControlHorizontalBackwards : BOOL;
	ResetMethodCallInitDriveMR01_Backwards : BOOL;
	ResetMethodCallInitDriveMR01_Forwards : BOOL;
END_VAR
VAR
	DirectionHorizontal : STRING;
	
	MBS_MR01_InitDrive_HorizontalForwards: AxisControl_MultipleInputSensors;
	MBS_MR01_InitDrive_HorizontalBackwards: AxisControl_MultipleInputSensors;
END_VAR

MBS_MR01_InitDrive_HorizontalBackwards(
    MethodCall := MethodCall_InitDrive,
    EmergencyStopSignal := ESS,
    Direction := DirectionHorizontal,
    InitStateDrive_Input := InputInitStateDrive,
    DI01 := ,
    DI02 := TouchSensor01,
    TouchSensorRelief := ,
    TOF_Time_MotorControl := ,
    TOF_Time_TouchSensorRelief := ,
    OperatingMode := InitDriveMode
);
MotorControlHorizontalBackwards := MBS_MR01_InitDrive_HorizontalBackwards.DigitalOutputControl_01;
MBS_MR01_InitDrive_HorizontalForwards(
    MethodCall := MethodCall_InitDrive,
    EmergencyStopSignal := ESS,
    Direction := DirectionHorizontal,
    InitStateDrive_Input := ,
    DI01 := TouchSensor01,
    DI02 := TouchSensor02,
    TouchSensorRelief := ,
    TOF_Time_MotorControl := ,
    TOF_Time_TouchSensorRelief := ,
    OperatingMode := InitDriveMode
);
MotorControlHorizontalForwards := MBS_MR01_InitDrive_HorizontalForwards.DigitalOutputControl_01;

END_FUNCTION_BLOCK

// ---- POUs/InitStateDrive/MBS_MR02_InitialStateDrive.TcPOU
FUNCTION_BLOCK MBS_MR02_InitialStateDrive
VAR_INPUT
	MethodCall_InitDrive : BOOL;
	ESS : BOOL;
	InputInitialStateDrive : BOOL;
	TOF_Time_InitCuttingTime : TIME;
	InitDriveMode : BOOL;
END_VAR
VAR_OUTPUT
	CheckMR02MotorControl : BOOL;
	ResetMethodCallCuttingProcess : BOOL;
END_VAR
VAR
	MBS_MR02_InitDrive_CuttingProcess: CuttingProcess;
END_VAR

MBS_MR02_InitDrive_CuttingProcess(
    MethodCall := MethodCall_InitDrive,
    EmergencyStopSignal := ESS,
    InitStateDrive_Input := InputInitialStateDrive,
    DI01 := ,
    TOF_Time_CuttingTime := TOF_Time_InitCuttingTime,
    OperatingMode := InitDriveMode
);
CheckMR02MotorControl := MBS_MR02_InitDrive_CuttingProcess.DigitalOutputControl_01;

END_FUNCTION_BLOCK

// ---- POUs/InitStateDrive/MBS_VSG_InitialStateDrive.TcPOU
FUNCTION_BLOCK MBS_VSG_InitialStateDrive
VAR_INPUT
	MethodCall_InitDrive : BOOL;
	ESS : BOOL;
	InputInitStateDrive : BOOL;
	TouchSensor01 : BOOL;
	TOF_Time_TSR : TIME;
	InitDriveMode : BOOL;	
END_VAR

VAR_OUTPUT
	DO_HorizontalMoveInitDriveVSG_01 : BOOL;
	DO_HorizontalMoveInitDriveVSG_02 : BOOL;
	ResetMethodCallInitDriveVSG : BOOL;
END_VAR

VAR
	TSR : BOOL := TRUE;
	DirectionHorizontal : STRING;

	MBS_VSG_InitDrive: AxisControl_MultipleInputSensors;
END_VAR

MBS_VSG_InitDrive(
    MethodCall := MethodCall_InitDrive,
    EmergencyStopSignal := ESS,
    Direction := DirectionHorizontal,
    InitStateDrive_Input := InputInitStateDrive,
    DI01 := ,
    DI02 := TouchSensor01,
    TouchSensorRelief := TSR,
    TOF_Time_MotorControl := ,
    TOF_Time_TouchSensorRelief := TOF_Time_TSR,
    OperatingMode := InitDriveMode
);
DO_HorizontalMoveInitDriveVSG_01 := MBS_VSG_InitDrive.DigitalOutputControl_01;

END_FUNCTION_BLOCK

// ---- POUs/InitStateDrive/SST_PD_InitialStateDrive.TcPOU
FUNCTION_BLOCK SST_PD_InitialStateDrive
VAR_INPUT
	MethodCall_InitDrive : BOOL;
	ESS : BOOL;
	InputInitialStateDrive : BOOL;
	TON_Time_PowerOFFSelfSet : TIME;
	InitDriveMode : BOOL;
END_VAR
VAR_OUTPUT
	MotorControl_PD01_Compressor : BOOL;
	MotorControl_PD01_Valve : BOOL;
	MotorControl_PD02_Compressor : BOOL;
	MotorControl_PD02_Valve : BOOL;
	MotorControl_PD03_Compressor : BOOL;
	MotorControl_PD03_Valve : BOOL;
	ResetMethodCallMovePD01 : BOOL;
	ResetMethodCallMovePD02 : BOOL;
	ResetMethodCallMovePD03 : BOOL;
END_VAR
VAR
	DestinationHorizontal : STRING;
	PowerOfF_SelfSet : BOOL := TRUE;
	SST_PD01_InitDrive : CompressorControl;
	SST_PD02_InitDrive : CompressorControl;
	SST_PD03_InitDrive : CompressorControl;
END_VAR

SST_PD01_InitDrive(
    MethodCall := MethodCall_InitDrive,
    EmergencyStopSignal := ESS,
    Destination := DestinationHorizontal,
    InitStateDrive_Input := InputInitialStateDrive,
    DI01 := ,
    DI02 := ,
    DI03_EncoderStart01 := ,
    DI04_EncoderStart02 := ,
    DI05_EncoderStart03 := ,
    DI06_EncoderStart04 := ,
    DI07_EncoderStart05 := ,
    DI08_EncoderStart06 := ,
    DI09_EncoderTarget01 := ,
    DI10_EncoderTarget02 := ,
    DI11_EncoderTarget03 := ,
    DI12_EncoderTarget04 := ,
    DI13_EncoderTarget05 := ,
    DI14_EncoderTarget06 := ,
    PowerOFF_SelfSet := PowerOfF_SelfSet,
    TON_Time_PowerOFFSelfSet := TON_Time_PowerOFFSelfSet,
    TON_Time_Compressor := PowerOnDelay_Compressor,
    TON_Time_Valve := PowerOnDelay_Valve,
    OperatingMode := AutomaticMode
);
MotorControl_PD01_Compressor := SST_PD01_InitDrive.DigitalOutputControl_01;
SST_PD02_InitDrive(
    MethodCall := MethodCall_InitDrive,
    EmergencyStopSignal := ESS,
    Destination := DestinationHorizontal,
    InitStateDrive_Input := InputInitialStateDrive,
    DI01 := ,
    DI02 := ,
    DI03_EncoderStart01 := ,
    DI04_EncoderStart02 := ,
    DI05_EncoderStart03 := ,
    DI06_EncoderStart04 := ,
    DI07_EncoderStart05 := ,
    DI08_EncoderStart06 := ,
    DI09_EncoderTarget01 := ,
    DI10_EncoderTarget02 := ,
    DI11_EncoderTarget03 := ,
    DI12_EncoderTarget04 := ,
    DI13_EncoderTarget05 := ,
    DI14_EncoderTarget06 := ,
    PowerOFF_SelfSet := PowerOfF_SelfSet,
    TON_Time_PowerOFFSelfSet := TON_Time_PowerOFFSelfSet,
    TON_Time_Compressor := PowerOnDelay_Compressor,
    TON_Time_Valve := PowerOnDelay_Valve,
    OperatingMode := AutomaticMode
);
MotorControl_PD02_Compressor := SST_PD02_InitDrive.DigitalOutputControl_01;
SST_PD03_InitDrive(
    MethodCall := MethodCall_InitDrive,
    EmergencyStopSignal := ESS,
    Destination := DestinationHorizontal,
    InitStateDrive_Input := InputInitialStateDrive,
    DI01 := ,
    DI02 := ,
    DI03_EncoderStart01 := ,
    DI04_EncoderStart02 := ,
    DI05_EncoderStart03 := ,
    DI06_EncoderStart04 := ,
    DI07_EncoderStart05 := ,
    DI08_EncoderStart06 := ,
    DI09_EncoderTarget01 := ,
    DI10_EncoderTarget02 := ,
    DI11_EncoderTarget03 := ,
    DI12_EncoderTarget04 := ,
    DI13_EncoderTarget05 := ,
    DI14_EncoderTarget06 := ,
    PowerOFF_SelfSet := PowerOfF_SelfSet,
    TON_Time_PowerOFFSelfSet := TON_Time_PowerOFFSelfSet,
    TON_Time_Compressor := PowerOnDelay_Compressor,
    TON_Time_Valve := PowerOnDelay_Valve,
    OperatingMode := AutomaticMode
);
MotorControl_PD03_Compressor := SST_PD03_InitDrive.DigitalOutputControl_01;

END_FUNCTION_BLOCK

// ---- POUs/MBS_SkillSet.TcPOU
PROGRAM MBS_SkillSet
VAR
//Multibearbeitungsstation Skills
	//MBS Maschine1 (Ofen) Skills	
	{attribute 'OPC.UA.DA':= '1'}
	MBS_Skill_MR01_TransportIn: MBS_MR01_AS_HorizontalMoveSensors;
	{attribute 'OPC.UA.DA':= '1'}
	MBS_Skill_MR01_SecuringWorkpiece: MBS_MR01_AS_SecuringProcess;
	{attribute 'OPC.UA.DA':= '1'}
	MBS_Skill_MR01_HardeningProcess: MBS_MR01_AS_HardeningProcess;
	{attribute 'OPC.UA.DA':= '1'}
	MBS_SkillMR01_ReleaseWorkpiece: MBS_MR01_AS_SecuringProcess;
	{attribute 'OPC.UA.DA':= '1'}
	MBS_Skill_MR01_TransportOut: MBS_MR01_AS_HorizontalMoveSensors;
	
	//MBS Vakuumsauggreifer Skills
	{attribute 'OPC.UA.DA':= '1'}
	MBS_Skill_VGS_PickUpWorkpieceToDmPD: MBS_VSG_AS_SuctionProcess;
	{attribute 'OPC.UA.DA':= '1'}
	MBS_Skill_VGS_PickUpWorkpieceToOven: MBS_VSG_AS_SuctionProcess;
	{attribute 'OPC.UA.DA':= '1'}
	MBS_Skill_VSG_VerticalMove: MBS_VSG_AS_VerticalMove;	
	{attribute 'OPC.UA.DA':= '1'}
	MBS_Skill_VSG_TransportToDmPD: MBS_VSG_AS_HorizontalMove;
	{attribute 'OPC.UA.DA':= '1'}
	MBS_Skill_VSG_TransportToMR01: MBS_VSG_AS_HorizontalMove;
	
	
	//MBS Drehteller mit PushingDevice Skills
	{attribute 'OPC.UA.DA':= '1'}
	MBS_Skill_DmPD_RotateFromVSGtoMR02: MBS_DmPD_AS_RotationMove;
	{attribute 'OPC.UA.DA':= '1'}
	MBS_Skill_DmPD_RotateFromVSGtoCB: MBS_DmPD_AS_RotationMove;
	{attribute 'OPC.UA.DA':= '1'}
	MBS_Skill_DmPD_RotateFromMR02toCB: MBS_DmPD_AS_RotationMove;
	{attribute 'OPC.UA.DA':= '1'}
	MBS_Skill_DmPD_RotateFromMR02toVSG: MBS_DmPD_AS_RotationMove;
	{attribute 'OPC.UA.DA':= '1'}
	MBS_Skill_DmPD_RotateFromCBtoVSG: MBS_DmPD_AS_RotationMove;
	{attribute 'OPC.UA.DA':= '1'}
	MBS_Skill_DmPD_RotateFromCBtoMR02: MBS_DmPD_AS_RotationMove;
	{attribute 'OPC.UA.DA':= '1'}
	MBS_Skill_DmPB_PushWorkpieceOff: MBS_DmPD_AS_HorizontalMove;
	
	//MBS Maschine2 (Schneidemaschine) Skills
	{attribute 'OPC.UA.DA':= '1'}
	MBS_Skill_MR02_CuttingProcess: MBS_MR02_AS_CuttingProcess;
	
	//MBS ConveyorBelt Skills
	{attribute 'OPC.UA.DA':= '1'}
	MBS_Skill_CB_Moving: MBS_CB_AS_HorizontalMove;
	
	//Organisation FBs
	MBS_ControlOfOutputs : MBS_ControlOfOutputs;
	MBS_OperatingModes : MBS_OperatingModes;
	
	//InitialStateDrives
	MBS_MR01_InitialStateDrive : MBS_MR01_InitialStateDrive;
	MBS_VSG_InitialStateDrive : MBS_VSG_InitialStateDrive;
	MBS_DmPD_InitialStateDrive : MBS_DmPD_InitialStateDrive;
	MBS_MR02_InitialStateDrive : MBS_MR02_InitialStateDrive;
	
//Variablen zur Outputsteuerung
	//Output-Variablen der Komponente MR01 
	MR01_MoveOvenslideIn 			: BOOL; //GVL_MBS.MBS_MOT_Ofenschieber_einfahren
	MR01_MoveOvenslideOut			: BOOL; //GVL_MBS.MBS_MOT_Ofenschieber_ausfahren
	MR01_Compressor_SecuringProcess : BOOL; //GVL_MBS.MBS_Kompressor
	MR01_Valve_OvenDoor				: BOOL; //GVL_MBS.MBS_MV_Ofentuer
	MR01_HardeningProcess			: BOOL; //GVL_MBS.MBS_Leuchte_Ofen
	
	//Output-Variablen der Komponente VSG
	VSG_Compressor_VerticalMove			: BOOL; //GVL_MBS.MBS_Kompressor
	VSG_Valve_VerticalMove				: BOOL; //GVL_MBS.MBS_MV_senken
	VSG_Compressor_SuctionProcessToDmPD	: BOOL; //GVL_MBS.MBS_Kompressor
	VSG_Valve_SuctionProcessToDmPD		: BOOL; //GVL_MBS.MBS_MV_Vakuum
	VSG_Compressor_SuctionProcessToMR01	: BOOL; //GVL_MBS.MBS_Kompressor
	VSG_Valve_SuctionProcessToMR01		: BOOL; //GVL_MBS.MBS_MV_Vakuum
	VSG_MoveHorizontalForwards			: BOOL; //GVL_MBS.MBS_MOT_Sauger_zum_DK
	VSG_MoveHorizontalBackwards			: BOOL; //GVL_MBS.MBS_MOT_Sauger_zum_Ofen
		
	//Output-Variablen der Komponente DmPD
	DmPD_RotateCWformVSGtoMR02 		: BOOL; //GVL_MBS.MBS_MOT_DK_CW
	DmPD_RotateCWromVSGtoCB			: BOOL; //GVL_MBS.MBS_MOT_DK_CW
	DmPD_RotateCWfromMR02toCB		: BOOL; //GVL_MBS.MBS_MOT_DK_CW
	DmPD_RotateCCWformCBtoMR02 		: BOOL; //GVL_MBS.MBS_MOT_DK_CCW
	DmPD_RotateCCWformCBtoVSG 		: BOOL; //GVL_MBS.MBS_MOT_DK_CCW
	DmPD_RotateCCWformMR02toVSG 	: BOOL; //GVL_MBS.MBS_MOT_DK_CCW
	DmPD_Compressor_HorizontalMove 	: BOOL; //GVL_MBS.MBS_Kompressor
	DmPD_Valve_HorizontalMove 		: BOOL; //GVL_MBS.ControlValveHorizontalMove
	
	//Output-Variablen der Komponente MR02
	MR02_CuttingProcess : BOOL; //GVL_MBS.MBS_MOT_Saege
	
	//Output-Variablen der Komponente CB
	CB_MoveForwards	: BOOL; //GVL_MBS.MBS_MOT_Foerderband_vorwaerts
	
//Output-Variablen für Init-Fahrt
	Init_MR01_HorizontalForwards	: BOOL; //GVL_MBS.MBS_MOT_Ofenschieber_einfahren
	Init_MR01_HorizontalBackwards	: BOOL; //GVL_MBS.MBS_MOT_Ofenschieber_ausfahren
	Init_VSG_HorizontalForwards 	: BOOL; //GVL_MBS.MBS_MOT_Sauger_zum_DK
	Init_VSG_HorizontalBackwards	: BOOL; //GVL_MBS.MBS_MOT_Sauger_zum_Ofen
	Init_DmPD_RotateCW				: BOOL; //GVL_MBS.MBS_MOT_DK_CW
	Init_DmPD_RotateCCW				: BOOL; //GVL_MBS.MBS_MOT_DK_CCW
	Init_MR02_CuttingProcess		: BOOL; //GVL_MBS.MBS_MOT_Saege
	
//Variablensetzung: Sollte später über SkillOA eingesetzt werden ODER Hard in SPS codiert (Diskussionspunkt)
	ResetButton: BOOL;
	StartButton: BOOL;
	ConfirmationButton: BOOL;

//Time Constraints
	TIME_TSR : TIME := T#150MS;
	PowerOnDelay_Compressor : TIME := T#500MS;
	PowerOnDelay_Valve_SuctionProcess : TIME := T#520MS;
	PowerOnDelay_Valve_VerticalMove : TIME := T#120MS;
	PowerOnDelay_Valve_HorizontalMove : TIME := T#120MS;
	PowerOffDelay_ConveyorBelt : TIME := T#100MS;	
//Encoder Values for InitialStateDrive
	
//Variable Values for InitialStateDrive
	MethodCall_InitStateDrive	: BOOL;
	InputVar_InitStateDrive		: BOOL;
	InitTime_Cutting 			: TIME := T#200MS;

END_VAR

MBS_OperatingModes(
    Start := StartButton,
    Stop := ((GVL.diNotAus_Kanal_A) AND (GVL.diNotAus_Kanal_B)),
    Reset := ResetButton,
    Schalter := ConfirmationButton,
    Schrittkette_GS := (((MBS_MR01_InitialStateDrive.ResetMethodCallInitDriveMR01_Backwards) AND (MBS_MR01_InitialStateDrive.ResetMethodCallInitDriveMR01_Forwards) AND (MBS_VSG_InitialStateDrive.ResetMethodCallInitDriveVSG) AND (MBS_DmPD_InitialStateDrive.ResetMethodCallRotateCCW) AND (MBS_DmPD_InitialStateDrive.ResetMethodCallRotateCW) AND (MBS_MR02_InitialStateDrive.ResetMethodCallCuttingProcess)))
);
MBS_ControlOfOutputs(
    F4 := MBS_OperatingModes.F4,
    F1 := MBS_OperatingModes.F1,
    A2 := MBS_OperatingModes.A2,
    A1 := MBS_OperatingModes.A1,
    A6 := MBS_OperatingModes.A6,
    Start := MBS_OperatingModes.Start,
    CB_Forwards := CB_MoveForwards,
    DmPD_Compressor := DmPD_Compressor_HorizontalMove,
    DmPD_Valve := DmPD_Valve_HorizontalMove,
    DmPD_RotateCW_VSGtoMR02 := DmPD_RotateCWformVSGtoMR02,
    DmPD_RotateCW_VSGtoCB := DmPD_RotateCWromVSGtoCB,
    DmPD_RotateCW_MR02toCB := DmPD_RotateCWfromMR02toCB,
    DmPD_RotateCCW_CBtoMR02 := DmPD_RotateCCWformCBtoMR02,
    DmPD_RotateCCW_CBtoVSG := DmPD_RotateCCWformCBtoVSG,
    DmPD_RotateCCW_MR02toVSG := DmPD_RotateCCWformMR02toVSG,
    MR01_HardeningProcess := MR01_HardeningProcess,
    MR01_HorizontalForwards := MR01_MoveOvenslideIn,
    MR01_HoritzontalBackwards := MR01_MoveOvenslideOut,
    MR01_Compressor := MR01_Compressor_SecuringProcess,
    MR01_Valve := MR01_Valve_OvenDoor,
    MR02_CuttingProcess := MR02_CuttingProcess,
    VSG_HorizontalForwards := VSG_MoveHorizontalForwards,
    VSG_HorizontalBackwards := VSG_MoveHorizontalBackwards,
    VSG_Valve_VerticalDown := VSG_Valve_VerticalMove,
    VSG_Valve_SuctionToDmPD := VSG_Valve_SuctionProcessToDmPD,
    VSG_Valve_SuctionToMR01 := VSG_Valve_SuctionProcessToMR01,
    VSG_Compressor_VerticalDown := VSG_Compressor_VerticalMove,
    VSG_Compressor_SuctionToDmPD := VSG_Compressor_SuctionProcessToDmPD,
    VSG_Compressor_SuctionToMR01 := VSG_Compressor_SuctionProcessToMR01,
    Init_DmPD_RotateCCW := Init_DmPD_RotateCCW,
    Init_DmPD_RotateCW := Init_DmPD_RotateCW,
    Init_MR01_HorizontalForwards := Init_MR01_HorizontalForwards,
    Init_MR01_HorizontalBackwards := Init_MR01_HorizontalBackwards,
    Init_MR02_CuttingProcess := Init_MR02_CuttingProcess,
    Init_VSG_HorizontalForwards := Init_VSG_HorizontalForwards,
    Init_VSG_HorizontalBackwards := Init_VSG_HorizontalBackwards
);
GVL_MBS.MBS_MOT_Foerderband_vorwaerts := MBS_ControlOfOutputs.ConveyorBeltForward;
MBS_MR01_InitialStateDrive(
    MethodCall_InitDrive := MethodCall_InitStateDrive,
    ESS := ((GVL.diNotAus_Kanal_A) AND (GVL.diNotAus_Kanal_B)),
    InputInitStateDrive := InputVar_InitStateDrive,
    TouchSensor01 := GVL_MBS.MBS_Ref_Taster_Ofenschieber_innen,
    TouchSensor02 := GVL_MBS.MBS_Ref_Taster_Ofenschieber_aussen,
    InitDriveMode := MBS_OperatingModes.A6
);
Init_MR01_HorizontalForwards := MBS_MR01_InitialStateDrive.MotorControlHorizontalForwards;
MBS_VSG_InitialStateDrive(
    MethodCall_InitDrive := MethodCall_InitStateDrive,
    ESS := ((GVL.diNotAus_Kanal_A) AND (GVL.diNotAus_Kanal_B)),
    InputInitStateDrive := InputVar_InitStateDrive,
    TouchSensor01 := GVL_MBS.MBS_Ref_Taster_Sauger_Pos_DK,
    TOF_Time_TSR := TIME_TSR,
    InitDriveMode := MBS_OperatingModes.A6
);
Init_VSG_HorizontalForwards := MBS_VSG_InitialStateDrive.DO_HorizontalMoveInitDriveVSG_01;
MBS_DmPD_InitialStateDrive(
    MethodCall_InitDrive := MethodCall_InitStateDrive,
    ESS := ((GVL.diNotAus_Kanal_A) AND (GVL.diNotAus_Kanal_B)),
    InputInitialStateDrive := InputVar_InitStateDrive,
    DI02_CW := GVL_MBS.MBS_Ref_Taster_DK_Pos_Foerderband,
    DI01_CCW := GVL_MBS.MBS_Ref_Taster_DK_Pos_Foerderband,
    DI02_CCW := GVL_MBS.MBS_Ref_Taster_DK_Pos_Sauger,
    InitDriveMode := MBS_OperatingModes.A6
);
Init_DmPD_RotateCW := MBS_DmPD_InitialStateDrive.MotorControl_CW;
MBS_MR02_InitialStateDrive(
    MethodCall_InitDrive := MethodCall_InitStateDrive,
    ESS := ((GVL.diNotAus_Kanal_A) AND (GVL.diNotAus_Kanal_B)),
    InputInitialStateDrive := InputVar_InitStateDrive,
    TOF_Time_InitCuttingTime := InitTime_Cutting,
    InitDriveMode := MBS_OperatingModes.A6
);
Init_MR02_CuttingProcess := MBS_MR02_InitialStateDrive.CheckMR02MotorControl;
MBS_Skill_MR01_TransportIn(
    ESS := ((GVL.diNotAus_Kanal_A) AND (GVL.diNotAus_Kanal_B)),
    TouchSensor_01 := GVL_MBS.MBS_Ref_Taster_Ofenschieber_aussen,
    TouchSensor_02 := GVL_MBS.MBS_Ref_Taster_Ofenschieber_innen,
    TOF_Time_TSR := TIME_TSR,
    AutomaticMode := MBS_OperatingModes.F1
);
MR01_MoveOvenslideIn := MBS_Skill_MR01_TransportIn.DO_MovingHorizontalMR01_01;
MBS_Skill_MR01_TransportOut(
    ESS := ((GVL.diNotAus_Kanal_A) AND (GVL.diNotAus_Kanal_B)),
    TouchSensor_01 := GVL_MBS.MBS_Ref_Taster_Ofenschieber_innen,
    TouchSensor_02 := GVL_MBS.MBS_Ref_Taster_Ofenschieber_aussen,
    TOF_Time_TSR := TIME_TSR,
    AutomaticMode := MBS_OperatingModes.F1
);
MR01_MoveOvenslideOut := MBS_Skill_MR01_TransportOut.DO_MovingHorizontalMR01_01;
MBS_Skill_MR01_SecuringWorkpiece(ESS := ((GVL.diNotAus_Kanal_A) AND (GVL.diNotAus_Kanal_B)), TouchSensor_01 := GVL_MBS.MBS_Ref_Taster_Ofenschieber_innen, AutomaticMode := MBS_OperatingModes.F1);
MR01_Compressor_SecuringProcess := MBS_Skill_MR01_SecuringWorkpiece.DO_SecuringProcessCompressorMR01_01;
MBS_Skill_MR01_HardeningProcess(ESS := ((GVL.diNotAus_Kanal_A) AND (GVL.diNotAus_Kanal_B)), LightSensor_01 := GVL_MBS.MBS_Ref_Taster_Ofenschieber_innen, AutomaticMode := MBS_OperatingModes.F1);
MR01_HardeningProcess := MBS_Skill_MR01_HardeningProcess.DO_HardeningProcessControlMR01;
MBS_Skill_VSG_VerticalMove(
    ESS := ((GVL.diNotAus_Kanal_A) AND (GVL.diNotAus_Kanal_B)),
    TouchSensor_01 := GVL_MBS.MBS_Ref_Taster_Sauger_Pos_DK,
    TON_PowerOnDelay_Compressor := PowerOnDelay_Compressor,
    TON_PowerOnDelay_Valve := PowerOnDelay_Valve_VerticalMove,
    AutomaticMode := MBS_OperatingModes.F1
);
VSG_Compressor_VerticalMove := MBS_Skill_VSG_VerticalMove.DO_ControlCompressorVerticalMoveVSG_01;
MBS_Skill_VGS_PickUpWorkpieceToDmPD(
    ESS := ((GVL.diNotAus_Kanal_A) AND (GVL.diNotAus_Kanal_B)),
    TouchSensor_01 := GVL_MBS.MBS_Ref_Taster_Sauger_Pos_Ofen,
    TouchSensor_02 := GVL_MBS.MBS_Ref_Taster_Sauger_Pos_DK,
    TON_PowerOnDelay_Compressor := PowerOnDelay_Compressor,
    TON_PowerOnDelay_Valve := PowerOnDelay_Valve_SuctionProcess,
    AutomaticMode := MBS_OperatingModes.F1
);
VSG_Compressor_SuctionProcessToDmPD := MBS_Skill_VGS_PickUpWorkpieceToDmPD.DO_ControlCompressorSuctionProcessVSG_01;
MBS_Skill_VGS_PickUpWorkpieceToOven(
    ESS := ((GVL.diNotAus_Kanal_A) AND (GVL.diNotAus_Kanal_B)),
    TouchSensor_01 := GVL_MBS.MBS_Ref_Taster_Sauger_Pos_DK,
    TouchSensor_02 := GVL_MBS.MBS_Ref_Taster_Sauger_Pos_Ofen,
    TON_PowerOnDelay_Compressor := PowerOnDelay_Compressor,
    TON_PowerOnDelay_Valve := PowerOnDelay_Valve_SuctionProcess,
    AutomaticMode := MBS_OperatingModes.F1
);
VSG_Compressor_SuctionProcessToMR01 := MBS_Skill_VGS_PickUpWorkpieceToOven.DO_ControlCompressorSuctionProcessVSG_01;
MBS_Skill_VSG_TransportToDmPD(
    ESS := ((GVL.diNotAus_Kanal_A) AND (GVL.diNotAus_Kanal_B)),
    TouchSensor_01 := GVL_MBS.MBS_Ref_Taster_Sauger_Pos_Ofen,
    TouchSensor_02 := GVL_MBS.MBS_Ref_Taster_Sauger_Pos_DK,
    TOF_Time_TSR := TIME_TSR,
    AutomaticeMode := MBS_OperatingModes.F1
);
VSG_MoveHorizontalForwards := MBS_Skill_VSG_TransportToDmPD.DO_HorizontalMoveVSG_01;
MBS_Skill_VSG_TransportToMR01(
    ESS := ((GVL.diNotAus_Kanal_A) AND (GVL.diNotAus_Kanal_B)),
    TouchSensor_01 := GVL_MBS.MBS_Ref_Taster_Sauger_Pos_DK,
    TouchSensor_02 := GVL_MBS.MBS_Ref_Taster_Sauger_Pos_Ofen,
    TOF_Time_TSR := TIME_TSR,
    AutomaticeMode := MBS_OperatingModes.F1
);
VSG_MoveHorizontalBackwards := MBS_Skill_VSG_TransportToMR01.DO_HorizontalMoveVSG_01;
MBS_Skill_DmPD_RotateFromVSGtoMR02(
    ESS := ((GVL.diNotAus_Kanal_A) AND (GVL.diNotAus_Kanal_B)),
    TouchSensor_01 := GVL_MBS.MBS_Ref_Taster_DK_Pos_Sauger,
    TouchSensor_02 := GVL_MBS.MBS_Ref_Taster_DK_Pos_Saege,
    AutomaticMode := MBS_OperatingModes.F1
);
DmPD_RotateCWformVSGtoMR02 := MBS_Skill_DmPD_RotateFromVSGtoMR02.DO_MovingRotationPmPD_01;
MBS_Skill_DmPD_RotateFromVSGtoCB(
    ESS := ((GVL.diNotAus_Kanal_A) AND (GVL.diNotAus_Kanal_B)),
    TouchSensor_01 := GVL_MBS.MBS_Ref_Taster_DK_Pos_Sauger,
    TouchSensor_02 := GVL_MBS.MBS_Ref_Taster_DK_Pos_Foerderband,
    AutomaticMode := MBS_OperatingModes.F1
);
DmPD_RotateCWromVSGtoCB := MBS_Skill_DmPD_RotateFromVSGtoCB.DO_MovingRotationPmPD_01;
MBS_Skill_DmPD_RotateFromMR02toCB(
    ESS := ((GVL.diNotAus_Kanal_A) AND (GVL.diNotAus_Kanal_B)),
    TouchSensor_01 := GVL_MBS.MBS_Ref_Taster_DK_Pos_Saege,
    TouchSensor_02 := GVL_MBS.MBS_Ref_Taster_DK_Pos_Foerderband,
    AutomaticMode := MBS_OperatingModes.F1
);
DmPD_RotateCWfromMR02toCB := MBS_Skill_DmPD_RotateFromMR02toCB.DO_MovingRotationPmPD_01;
MBS_Skill_DmPD_RotateFromCBtoMR02(
    ESS := ((GVL.diNotAus_Kanal_A) AND (GVL.diNotAus_Kanal_B)),
    TouchSensor_01 := GVL_MBS.MBS_Ref_Taster_DK_Pos_Foerderband,
    TouchSensor_02 := GVL_MBS.MBS_Ref_Taster_DK_Pos_Saege,
    AutomaticMode := MBS_OperatingModes.F1
);
DmPD_RotateCCWformCBtoMR02 := MBS_Skill_DmPD_RotateFromCBtoMR02.DO_MovingRotationPmPD_01;
MBS_Skill_DmPD_RotateFromCBtoVSG(
    ESS := ((GVL.diNotAus_Kanal_A) AND (GVL.diNotAus_Kanal_B)),
    TouchSensor_01 := GVL_MBS.MBS_Ref_Taster_DK_Pos_Foerderband,
    TouchSensor_02 := GVL_MBS.MBS_Ref_Taster_DK_Pos_Sauger,
    AutomaticMode := MBS_OperatingModes.F1
);
DmPD_RotateCCWformCBtoVSG := MBS_Skill_DmPD_RotateFromCBtoVSG.DO_MovingRotationPmPD_01;
MBS_Skill_DmPD_RotateFromMR02toVSG(
    ESS := ((GVL.diNotAus_Kanal_A) AND (GVL.diNotAus_Kanal_B)),
    TouchSensor_01 := GVL_MBS.MBS_Ref_Taster_DK_Pos_Saege,
    TouchSensor_02 := GVL_MBS.MBS_Ref_Taster_DK_Pos_Sauger,
    AutomaticMode := MBS_OperatingModes.F1
);
DmPD_RotateCCWformMR02toVSG := MBS_Skill_DmPD_RotateFromMR02toVSG.DO_MovingRotationPmPD_01;
MBS_Skill_DmPB_PushWorkpieceOff(
    ESS := ((GVL.diNotAus_Kanal_A) AND (GVL.diNotAus_Kanal_B)),
    TouchSensor_01 := GVL_MBS.MBS_Ref_Taster_DK_Pos_Foerderband,
    TON_PowerOnDelay_Compressor := PowerOnDelay_Compressor,
    TON_PowerOnDelay_Valve := PowerOnDelay_Valve_HorizontalMove,
    AutomaticMode := MBS_OperatingModes.F1
);
DmPD_Compressor_HorizontalMove := MBS_Skill_DmPB_PushWorkpieceOff.DO_ControlCompressorDmPD_01;
MBS_Skill_MR02_CuttingProcess(ESS := ((GVL.diNotAus_Kanal_A) AND (GVL.diNotAus_Kanal_B)), TouchSensor_01 := GVL_MBS.MBS_Ref_Taster_DK_Pos_Saege, AutomaticMode := MBS_OperatingModes.F1);
MR02_CuttingProcess := MBS_Skill_MR02_CuttingProcess.DO_CuttingProcessControlMR02;
MBS_Skill_CB_Moving(
    ESS := ((GVL.diNotAus_Kanal_A) AND (GVL.diNotAus_Kanal_B)),
    TouchSensor_01 := GVL_MBS.MBS_Ref_Taster_DK_Pos_Foerderband,
    LightSensor_01 := GVL_MBS.MBS_LS_Ende_Foerderband,
    TOF_Time_MotorControl := PowerOffDelay_ConveyorBelt,
    AutomaticMode := MBS_OperatingModes.F1
);
CB_MoveForwards := MBS_Skill_CB_Moving.DO_MovingHorizontalCB_01;

END_PROGRAM

// ---- POUs/Moduls/MBS_Skills/MBS_MR01_AS_HorizontalMoveSensors.TcPOU
{attribute 'OPC.UA.DA.JobMethod' := 'JobMethode_HorizontalMove'}
FUNCTION_BLOCK MBS_MR01_AS_HorizontalMoveSensors
VAR
	AlwaysTrue : BOOL := TRUE;
	// Used for debugging purposes to display InputArguments of method call
	MethodCall_HorizontalMove : BOOL := FALSE; // used to store InputArg "MethodCall" from Start() method
	ResetMethodCall : BOOL := FALSE;
	DirectionHorizontal : STRING; // defines movement direction
	TSR : BOOL; // Variable that is needed to perform the relief of the touch sensor
	callCounterStart : ULINT; // counts how many times the Start() method has been called
	callCounterCheckState : ULINT; // counts how many times the CheckState() method has been called
	callCounterAbort : ULINT; // counts how many times the Abort() method has been called
	
	// Variables to determine if a job has been started (Start() method has been called) or finished
	jobRunning : BOOL;
	jobFinished : BOOL;

	// State machine variable
	state : UDINT;
	
	//Variablen des Transport FBs
	MBS_MR01_HorizontalMove : AxisControl_MultipleInputSensors;
END_VAR
	
VAR_INPUT
	ESS: BOOL;
	TouchSensor_01 : BOOL;
	TouchSensor_02 : BOOL;
	TOF_Time_TSR : TIME;
	AutomaticMode : BOOL;
END_VAR

VAR_OUTPUT
	DO_MovingHorizontalMR01_01 : BOOL;
	DO_MovingHorizontalMR01_02 : BOOL;
END_VAR

(* ST implementation auto-generated from FBD in export.xml *)
MBS_MR01_HorizontalMove(
    MethodCall := MethodCall_HorizontalMove,
    EmergencyStopSignal := ESS,
    Direction := DirectionHorizontal,
    InitStateDrive_Input := ,
    DI01 := TouchSensor_01,
    DI02 := TouchSensor_02,
    TouchSensorRelief := TSR,
    TOF_Time_MotorControl := ,
    TOF_Time_TouchSensorRelief := TOF_Time_TSR,
    OperatingMode := AutomaticMode
);
DO_MovingHorizontalMR01_01 := MBS_MR01_HorizontalMove.DigitalOutputControl_01;

{attribute 'TcRpcEnable' := '1'}
METHOD Abort : HRESULT
VAR_INPUT
	hdl : UDINT; // Do not change, used by server.
END_VAR
callCounterAbort := callCounterAbort + 1;
END_METHOD

{attribute 'TcRpcEnable' := '1'}
METHOD CheckState : HRESULT
VAR_INPUT
	hdl : UDINT; // Do not change, used by server.
END_VAR
VAR_OUTPUT
	bBusy : BOOL; // Do not change. Used by server to find out if the job is finished
	
	// List of OutputArguments for OPC UA method, may be customized
	State : BOOL; // Abgeschlossener MethodCall
	MethodCall: BOOL; //Input Recall
END_VAR
callCounterCheckState := callCounterCheckState + 1;
IF NOT jobFinished THEN
	bBusy := TRUE; // job is not finished yet
	CheckState := 0; // no error
ELSE
	bBusy := FALSE; // job is finished
	CheckState := 0; // done, no error occured during execution (OPC UA StatusCode "GOOD")
	jobFinished := FALSE;
	State := ResetMethodCall;
	MethodCall := MethodCall_HorizontalMove;
END_IF
END_METHOD

{attribute 'TcRpcEnable' := '1'}
METHOD Start : HRESULT
VAR_INPUT
	// List of InputArguments for OPC UA method, may be customized
	MethodCall : BOOL; // some description
	ProcessingTime : TIME;
END_VAR
VAR_OUTPUT
	hdl : UDINT; // Do not change, used by server.
END_VAR
callCounterStart := callCounterStart + 1;

MethodCall_HardeningProcess := MethodCall;
ProcessingTime_HardeningProcess := ProcessingTime;

jobRunning := TRUE;
Start := 0; // no error occured, e.g. while parsing the input arguments (0 = OPC UA StatusCode "GOOD")
END_METHOD

END_FUNCTION_BLOCK

// ---- POUs/Moduls/MBS_Skills/MBS_MR01_AS_SecuringProcess.TcPOU
{attribute 'OPC.UA.DA.JobMethod' := 'JobMethode_SecuringProcess'}
FUNCTION_BLOCK MBS_MR01_AS_SecuringProcess
VAR
	AlwaysTrue : BOOL := TRUE;
	// Used for debugging purposes to display InputArguments of method call
	MethodCall_SecuringProcess : BOOL := FALSE; // used to store InputArg "MethodCall" from Start() method
	ResetMethodCall	: BOOL := FALSE;	
	SecuringTime : TIME;	//Time for Securing the Workpiece
	SecuringProcessingTime : TIME; //Two Times for Securing the Workpiece (for Secure and Release) + HardeningProcessingTime
	callCounterStart : ULINT; // counts how many times the Start() method has been called
	callCounterCheckState : ULINT; // counts how many times the CheckState() method has been called
	callCounterAbort : ULINT; // counts how many times the Abort() method has been called
	
	// Variables to determine if a job has been started (Start() method has been called) or finished
	jobRunning : BOOL;
	jobFinished : BOOL;

	// State machine variable
	state : UDINT;
	
	//Variablen des FBs
	MBS_MR01_SecuringProcess : SecuringWorkpiece;
END_VAR
	
VAR_INPUT
	ESS: BOOL;
	TouchSensor_01 : BOOL;
	AutomaticMode: BOOL;
END_VAR

VAR_OUTPUT
	DO_SecuringProcessCompressorMR01_01 : BOOL;
	DO_SecuringProcessValveMR01_02 : BOOL;
END_VAR

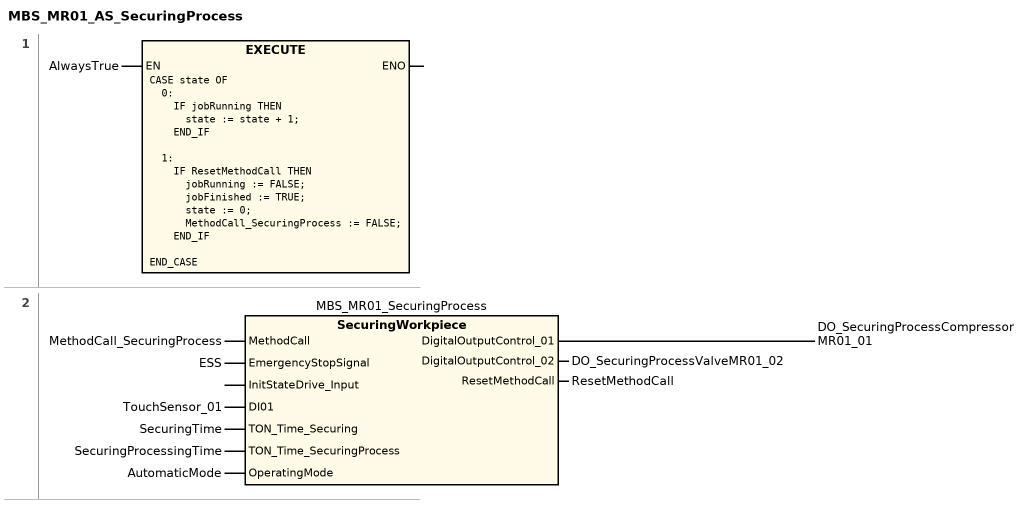
// NETWORK 1
IF AlwaysTrue THEN
    CASE state OF
    	0:
    		IF jobRunning THEN
    			state := state + 1;
    		END_IF
    		
    	1:
    		IF ResetMethodCall THEN
    			jobRunning := FALSE;
    			jobFinished := TRUE;
    			state := 0;
    			MethodCall_SecuringProcess := FALSE;
    		END_IF
    		
    END_CASE
END_IF

// NETWORK 2
MBS_MR01_SecuringProcess(
    MethodCall := MethodCall_SecuringProcess,
    EmergencyStopSignal := ESS,
    DI01 := TouchSensor_01,
    TON_Time_Securing := SecuringTime,
    TON_Time_SecuringProcess := SecuringProcessingTime,
    OperatingMode := AutomaticMode,
    DigitalOutputControl_02 => DO_SecuringProcessValveMR01_02,
    ResetMethodCall => ResetMethodCall); // SecuringWorkpiece
DO_SecuringProcessCompressorMR01_01 := MBS_MR01_SecuringProcess.DigitalOutputControl_01;

{attribute 'TcRpcEnable' := '1'}
METHOD Abort : HRESULT
VAR_INPUT
	hdl : UDINT; // Do not change, used by server.
END_VAR
callCounterAbort := callCounterAbort + 1;
END_METHOD

{attribute 'TcRpcEnable' := '1'}
METHOD CheckState : HRESULT
VAR_INPUT
	hdl : UDINT; // Do not change, used by server.
END_VAR
VAR_OUTPUT
	bBusy : BOOL; // Do not change. Used by server to find out if the job is finished
	
	// List of OutputArguments for OPC UA method, may be customized
	State : BOOL; // Abgeschlossener MethodCall
	MethodCall: BOOL; //Input Recall
END_VAR
callCounterCheckState := callCounterCheckState + 1;
IF NOT jobFinished THEN
	bBusy := TRUE; // job is not finished yet
	CheckState := 0; // no error
ELSE
	bBusy := FALSE; // job is finished
	CheckState := 0; // done, no error occured during execution (OPC UA StatusCode "GOOD")
	jobFinished := FALSE;
	State := ResetMethodCall;
	MethodCall := MethodCall_SecuringProcess;
END_IF
END_METHOD

{attribute 'TcRpcEnable' := '1'}
METHOD Start : HRESULT
VAR_INPUT
	// List of InputArguments for OPC UA method, may be customized
	MethodCall : BOOL; // some description
	Securing_Time : TIME;
	SecuringProcessing_Time : TIME;
END_VAR
VAR_OUTPUT
	hdl : UDINT; // Do not change, used by server.
END_VAR
callCounterStart := callCounterStart + 1;

MethodCall_SecuringProcess := MethodCall;
SecuringTime := Securing_Time;
SecuringProcessingTime := SecuringProcessing_Time;

jobRunning := TRUE;
Start := 0; // no error occured, e.g. while parsing the input arguments (0 = OPC UA StatusCode "GOOD")
END_METHOD

END_FUNCTION_BLOCK

// ---- POUs/Moduls/MBS_Skills/MBS_MR01_AS_HardeningProcess.TcPOU
{attribute 'OPC.UA.DA.JobMethod' := 'JobMethode_HardeningProcess'}
FUNCTION_BLOCK MBS_MR01_AS_HardeningProcess
VAR
	AlwaysTrue : BOOL := TRUE;
	// Used for debugging purposes to display InputArguments of method call
	MethodCall_HardeningProcess : BOOL := FALSE; // used to store InputArg "MethodCall" from Start() method
	ResetMethodCall	: BOOL := FALSE;
	ProcessingTime_HardeningProcess : TIME;
	callCounterStart : ULINT; // counts how many times the Start() method has been called
	callCounterCheckState : ULINT; // counts how many times the CheckState() method has been called
	callCounterAbort : ULINT; // counts how many times the Abort() method has been called
	
	// Variables to determine if a job has been started (Start() method has been called) or finished
	jobRunning : BOOL;
	jobFinished : BOOL;

	// State machine variable
	state : UDINT;
	
	//Variablen des FBs
	MBS_MR01_HardeningProcess : HardeningProcess;
END_VAR
	
VAR_INPUT
	ESS: BOOL;
	LightSensor_01 : BOOL;
	AutomaticMode : BOOL;
END_VAR

VAR_OUTPUT
	DO_HardeningProcessControlMR01 : BOOL;
END_VAR

MBS_MR01_HardeningProcess(
    MethodCall := MethodCall_HardeningProcess,
    EmergencyStopSignal := ESS,
    InitStateDrive_Input := ,
    DI01 := LightSensor_01,
    TOF_Time_HardeningTime := ProcessingTime_HardeningProcess,
    OperatingMode := AutomaticMode
);
DO_HardeningProcessControlMR01 := MBS_MR01_HardeningProcess.DigitalOutputControl_01;

{attribute 'TcRpcEnable' := '1'}
METHOD Abort : HRESULT
VAR_INPUT
	hdl : UDINT; // Do not change, used by server.
END_VAR
callCounterAbort := callCounterAbort + 1;
END_METHOD

{attribute 'TcRpcEnable' := '1'}
METHOD CheckState : HRESULT
VAR_INPUT
	hdl : UDINT; // Do not change, used by server.
END_VAR
VAR_OUTPUT
	bBusy : BOOL; // Do not change. Used by server to find out if the job is finished
	
	// List of OutputArguments for OPC UA method, may be customized
	State : BOOL; // Abgeschlossener MethodCall
	MethodCall: BOOL; //Input Recall
END_VAR
callCounterCheckState := callCounterCheckState + 1;
IF NOT jobFinished THEN
	bBusy := TRUE; // job is not finished yet
	CheckState := 0; // no error
ELSE
	bBusy := FALSE; // job is finished
	CheckState := 0; // done, no error occured during execution (OPC UA StatusCode "GOOD")
	jobFinished := FALSE;
	State := ResetMethodCall;
	MethodCall := MethodCall_HardeningProcess;
END_IF
END_METHOD

{attribute 'TcRpcEnable' := '1'}
METHOD Start : HRESULT
VAR_INPUT
	// List of InputArguments for OPC UA method, may be customized
	MethodCall : BOOL; // some description
	ProcessingTime : TIME;
END_VAR
VAR_OUTPUT
	hdl : UDINT; // Do not change, used by server.
END_VAR
callCounterStart := callCounterStart + 1;

MethodCall_HardeningProcess := MethodCall;
ProcessingTime_HardeningProcess := ProcessingTime;

jobRunning := TRUE;
Start := 0; // no error occured, e.g. while parsing the input arguments (0 = OPC UA StatusCode "GOOD")
END_METHOD

END_FUNCTION_BLOCK

// ---- POUs/Moduls/MBS_Skills/MBS_VSG_AS_SuctionProcess.TcPOU
{attribute 'OPC.UA.DA.JobMethod' := 'JobMethode_CompressorControl'}
FUNCTION_BLOCK MBS_VSG_AS_SuctionProcess
VAR
	AlwaysTrue : BOOL := TRUE;
	// Used for debugging purposes to display InputArguments of method call
	MethodCall_CompressorControl : BOOL := FALSE; // used to store InputArg "MethodCall" from Start() method
	ResetMethodCall	: BOOL := FALSE;
	Destination : STRING;
	callCounterStart : ULINT; // counts how many times the Start() method has been called
	callCounterCheckState : ULINT; // counts how many times the CheckState() method has been called
	callCounterAbort : ULINT; // counts how many times the Abort() method has been called
	
	// Variables to determine if a job has been started (Start() method has been called) or finished
	jobRunning : BOOL;
	jobFinished : BOOL;

	// State machine variable
	state : UDINT;
	
	//Variablen des Transport FBs
	MBS_VSG_SuctionProcess : CompressorControl;
END_VAR
	
VAR_INPUT
	ESS: BOOL;
	TouchSensor_01 : BOOL;
	TouchSensor_02 : BOOL;
	TON_PowerOnDelay_Compressor : TIME;
	TON_PowerOnDelay_Valve : TIME;
	AutomaticMode: BOOL;
END_VAR

VAR_OUTPUT
	DO_ControlCompressorSuctionProcessVSG_01 : BOOL;
	DO_ControlValveSuctionProcessVSG_02 : BOOL;
END_VAR

MBS_VSG_SuctionProcess(
    MethodCall := MethodCall_CompressorControl,
    EmergencyStopSignal := ESS,
    Destination := Destination,
    InitStateDrive_Input := ,
    DI01 := TouchSensor_01,
    DI02 := TouchSensor_02,
    DI03_EncoderStart01 := ,
    DI04_EncoderStart02 := ,
    DI05_EncoderStart03 := ,
    DI06_EncoderStart04 := ,
    DI07_EncoderStart05 := ,
    DI08_EncoderStart06 := ,
    DI09_EncoderTarget01 := ,
    DI10_EncoderTarget02 := ,
    DI11_EncoderTarget03 := ,
    DI12_EncoderTarget04 := ,
    DI13_EncoderTarget05 := ,
    DI14_EncoderTarget06 := ,
    PowerOFF_SelfSet := ,
    TON_Time_PowerOFFSelfSet := ,
    TON_Time_Compressor := TON_PowerOnDelay_Compressor,
    TON_Time_Valve := TON_PowerOnDelay_Valve,
    OperatingMode := AutomaticMode
);
DO_ControlCompressorSuctionProcessVSG_01 := MBS_VSG_SuctionProcess.DigitalOutputControl_01;

{attribute 'TcRpcEnable' := '1'}
METHOD Abort : HRESULT
VAR_INPUT
	hdl : UDINT; // Do not change, used by server.
END_VAR
callCounterAbort := callCounterAbort + 1;
END_METHOD

{attribute 'TcRpcEnable' := '1'}
METHOD CheckState : HRESULT
VAR_INPUT
	hdl : UDINT; // Do not change, used by server.
END_VAR
VAR_OUTPUT
	bBusy : BOOL; // Do not change. Used by server to find out if the job is finished
	
	// List of OutputArguments for OPC UA method, may be customized
	State : BOOL; // Abgeschlossener MethodCall
	MethodCall: BOOL; //Input Recall
END_VAR
callCounterCheckState := callCounterCheckState + 1;
IF NOT jobFinished THEN
	bBusy := TRUE; // job is not finished yet
	CheckState := 0; // no error
ELSE
	bBusy := FALSE; // job is finished
	CheckState := 0; // done, no error occured during execution (OPC UA StatusCode "GOOD")
	jobFinished := FALSE;
	State := ResetMethodCall;
	MethodCall := MethodCall_CompressorControl;
END_IF
END_METHOD

{attribute 'TcRpcEnable' := '1'}
METHOD Start : HRESULT
VAR_INPUT
	// List of InputArguments for OPC UA method, may be customized
	MethodCall : BOOL; // some description
	DestinationPoint : STRING;	
END_VAR
VAR_OUTPUT
	hdl : UDINT; // Do not change, used by server.
END_VAR
callCounterStart := callCounterStart + 1;

MethodCall_CompressorControl := MethodCall;
Destination := DestinationPoint;

jobRunning := TRUE;
Start := 0; // no error occured, e.g. while parsing the input arguments (0 = OPC UA StatusCode "GOOD")
END_METHOD

END_FUNCTION_BLOCK

// ---- POUs/Moduls/MBS_Skills/MBS_VSG_AS_VerticalMove.TcPOU
{attribute 'OPC.UA.DA.JobMethod' := 'JobMethode_CompressorControl'}
FUNCTION_BLOCK MBS_VSG_AS_VerticalMove
VAR
	AlwaysTrue : BOOL := TRUE;
	// Used for debugging purposes to display InputArguments of method call
	MethodCall_CompressorControl : BOOL := FALSE; // used to store InputArg "MethodCall" from Start() method
	ResetMethodCall	: BOOL := FALSE;
	DestinationVertical : STRING;
	PowerOFF_SelfSet : BOOL;
	PowerOFFDelay_SelfSet : TIME;
	callCounterStart : ULINT; // counts how many times the Start() method has been called
	callCounterCheckState : ULINT; // counts how many times the CheckState() method has been called
	callCounterAbort : ULINT; // counts how many times the Abort() method has been called
	
	// Variables to determine if a job has been started (Start() method has been called) or finished
	jobRunning : BOOL;
	jobFinished : BOOL;

	// State machine variable
	state : UDINT;
	
	//Variablen des Transport FBs
	MBS_VSG_VerticalMove : CompressorControl;
END_VAR
	
VAR_INPUT
	ESS: BOOL;
	TouchSensor_01 : BOOL;
	TON_PowerOnDelay_Compressor : TIME;
	TON_PowerOnDelay_Valve : TIME;
	AutomaticMode: BOOL;
END_VAR

VAR_OUTPUT
	DO_ControlCompressorVerticalMoveVSG_01 : BOOL;
	DO_ControlValveVerticalMoveVSG_02 : BOOL;
END_VAR

MBS_VSG_VerticalMove(
    MethodCall := MethodCall_CompressorControl,
    EmergencyStopSignal := ESS,
    Destination := DestinationVertical,
    InitStateDrive_Input := ,
    DI01 := TouchSensor_01,
    DI02 := ,
    DI03_EncoderStart01 := ,
    DI04_EncoderStart02 := ,
    DI05_EncoderStart03 := ,
    DI06_EncoderStart04 := ,
    DI07_EncoderStart05 := ,
    DI08_EncoderStart06 := ,
    DI09_EncoderTarget01 := ,
    DI10_EncoderTarget02 := ,
    DI11_EncoderTarget03 := ,
    DI12_EncoderTarget04 := ,
    DI13_EncoderTarget05 := ,
    DI14_EncoderTarget06 := ,
    PowerOFF_SelfSet := PowerOFF_SelfSet,
    TON_Time_PowerOFFSelfSet := PowerOFFDelay_SelfSet,
    TON_Time_Compressor := TON_PowerOnDelay_Compressor,
    TON_Time_Valve := TON_PowerOnDelay_Valve,
    OperatingMode := AutomaticMode
);
DO_ControlCompressorVerticalMoveVSG_01 := MBS_VSG_VerticalMove.DigitalOutputControl_01;

{attribute 'TcRpcEnable' := '1'}
METHOD Abort : HRESULT
VAR_INPUT
	hdl : UDINT; // Do not change, used by server.
END_VAR
callCounterAbort := callCounterAbort + 1;
END_METHOD

{attribute 'TcRpcEnable' := '1'}
METHOD CheckState : HRESULT
VAR_INPUT
	hdl : UDINT; // Do not change, used by server.
END_VAR
VAR_OUTPUT
	bBusy : BOOL; // Do not change. Used by server to find out if the job is finished
	
	// List of OutputArguments for OPC UA method, may be customized
	State : BOOL; // Abgeschlossener MethodCall
	MethodCall: BOOL; //Input Recall
END_VAR
callCounterCheckState := callCounterCheckState + 1;
IF NOT jobFinished THEN
	bBusy := TRUE; // job is not finished yet
	CheckState := 0; // no error
ELSE
	bBusy := FALSE; // job is finished
	CheckState := 0; // done, no error occured during execution (OPC UA StatusCode "GOOD")
	jobFinished := FALSE;
	State := ResetMethodCall;
	MethodCall := MethodCall_CompressorControl;
END_IF
END_METHOD

{attribute 'TcRpcEnable' := '1'}
METHOD Start : HRESULT
VAR_INPUT
	// List of InputArguments for OPC UA method, may be customized
	MethodCall : BOOL; // some description
	DestinationPoint : STRING;
	SelfSetPowerOff : BOOL;
	SelfSetPowerOffDelay : TIME;	
END_VAR
VAR_OUTPUT
	hdl : UDINT; // Do not change, used by server.
END_VAR
callCounterStart := callCounterStart + 1;

MethodCall_CompressorControl := MethodCall;
DestinationVertical := DestinationPoint;
PowerOFF_SelfSet := SelfSetPowerOff;
PowerOFFDelay_SelfSet := SelfSetPowerOffDelay;

jobRunning := TRUE;
Start := 0; // no error occured, e.g. while parsing the input arguments (0 = OPC UA StatusCode "GOOD")
END_METHOD

END_FUNCTION_BLOCK

// ---- POUs/Moduls/MBS_Skills/MBS_VSG_AS_HorizontalMove.TcPOU
{attribute 'OPC.UA.DA.JobMethod' := 'JobMethode_HorizontalMove'}
FUNCTION_BLOCK MBS_VSG_AS_HorizontalMove
VAR
	AlwaysTrue : BOOL := TRUE;
	// Used for debugging purposes to display InputArguments of method call
	MethodCall_HorizontalMove : BOOL := FALSE; // used to store InputArg "MethodCall" from Start() method
	ResetMethodCall	: BOOL := FALSE;
	DirectionHorizontal : STRING; // defines movement direction
	TSR : BOOL;// Variable that is needed to perform the relief of the touch sensor
	callCounterStart : ULINT; // counts how many times the Start() method has been called
	callCounterCheckState : ULINT; // counts how many times the CheckState() method has been called
	callCounterAbort : ULINT; // counts how many times the Abort() method has been called
	
	// Variables to determine if a job has been started (Start() method has been called) or finished
	jobRunning : BOOL;
	jobFinished : BOOL;

	// State machine variable
	state : UDINT;
	
	//Variablen des Transport FBs
	MBS_VSG_HorizontalMove : AxisControl_MultipleInputSensors;
END_VAR
	
VAR_INPUT
	ESS: BOOL;
	TouchSensor_01 : BOOL;
	TouchSensor_02 : BOOL;
	TOF_Time_TSR : TIME;
	AutomaticeMode : BOOL;
END_VAR

VAR_OUTPUT
	DO_HorizontalMoveVSG_01 : BOOL;
	DO_HorizontalMoveVSG_02 : BOOL;
END_VAR

MBS_VSG_HorizontalMove(
    MethodCall := MethodCall_HorizontalMove,
    EmergencyStopSignal := ESS,
    Direction := DirectionHorizontal,
    InitStateDrive_Input := ,
    DI01 := TouchSensor_01,
    DI02 := TouchSensor_02,
    TouchSensorRelief := TSR,
    TOF_Time_MotorControl := ,
    TOF_Time_TouchSensorRelief := TOF_Time_TSR,
    OperatingMode := AutomaticeMode
);
DO_HorizontalMoveVSG_01 := MBS_VSG_HorizontalMove.DigitalOutputControl_01;

{attribute 'TcRpcEnable' := '1'}
METHOD Abort : HRESULT
VAR_INPUT
	hdl : UDINT; // Do not change, used by server.
END_VAR
callCounterAbort := callCounterAbort + 1;
END_METHOD

{attribute 'TcRpcEnable' := '1'}
METHOD CheckState : HRESULT
VAR_INPUT
	hdl : UDINT; // Do not change, used by server.
END_VAR
VAR_OUTPUT
	bBusy : BOOL; // Do not change. Used by server to find out if the job is finished
	
	// List of OutputArguments for OPC UA method, may be customized
	State : BOOL; // Abgeschlossener MethodCall
	MethodCall: BOOL; //Input Recall
END_VAR
callCounterCheckState := callCounterCheckState + 1;
IF NOT jobFinished THEN
	bBusy := TRUE; // job is not finished yet
	CheckState := 0; // no error
ELSE
	bBusy := FALSE; // job is finished
	CheckState := 0; // done, no error occured during execution (OPC UA StatusCode "GOOD")
	jobFinished := FALSE;
	State := ResetMethodCall;
	MethodCall := MethodCall_HorizontalMove;
END_IF
END_METHOD

{attribute 'TcRpcEnable' := '1'}
METHOD Start : HRESULT
VAR_INPUT
	// List of InputArguments for OPC UA method, may be customized
	MethodCall : BOOL; // some description
	DirectionPoint : STRING;
	TouchSensorRelief : BOOL;	
END_VAR
VAR_OUTPUT
	hdl : UDINT; // Do not change, used by server.
END_VAR
callCounterStart := callCounterStart + 1;

MethodCall_HorizontalMove := MethodCall;
DirectionHorizontal := DirectionPoint;
TSR := TouchSensorRelief;

jobRunning := TRUE;
Start := 0; // no error occured, e.g. while parsing the input arguments (0 = OPC UA StatusCode "GOOD")
END_METHOD

END_FUNCTION_BLOCK

// ---- POUs/Moduls/MBS_Skills/MBS_DmPD_AS_RotationMove.TcPOU
{attribute 'OPC.UA.DA.JobMethod' := 'JobMethode_RotationMove'}
FUNCTION_BLOCK MBS_DmPD_AS_RotationMove
VAR
	AlwaysTrue : BOOL := TRUE;
	// Used for debugging purposes to display InputArguments of method call
	MethodCall_RotationMove : BOOL := FALSE; // used to store InputArg "MethodCall" from Start() method
	ResetMethodCall : BOOL := FALSE;
	DirectionRotation : STRING;
	callCounterStart : ULINT; // counts how many times the Start() method has been called
	callCounterCheckState : ULINT; // counts how many times the CheckState() method has been called
	callCounterAbort : ULINT; // counts how many times the Abort() method has been called
	
	// Variables to determine if a job has been started (Start() method has been called) or finished
	jobRunning : BOOL;
	jobFinished : BOOL;

	// State machine variable
	state : UDINT;
	
	//Variablen des Transport FBs
	MBS_DmPD_RotationMove : AxisControl_MultipleInputSensors;
END_VAR
	
VAR_INPUT
	ESS: BOOL;
	TouchSensor_01 : BOOL;
	TouchSensor_02 : BOOL;
	AutomaticMode: BOOL;
END_VAR

VAR_OUTPUT
	DO_MovingRotationPmPD_01 : BOOL;
	DO_MovingRotationPmPD_02 : BOOL;
END_VAR

MBS_DmPD_RotationMove(
    MethodCall := MethodCall_RotationMove,
    EmergencyStopSignal := ESS,
    Direction := DirectionRotation,
    InitStateDrive_Input := ,
    DI01 := TouchSensor_01,
    DI02 := TouchSensor_02,
    TouchSensorRelief := ,
    TOF_Time_MotorControl := ,
    TOF_Time_TouchSensorRelief := ,
    OperatingMode := AutomaticMode
);
DO_MovingRotationPmPD_01 := MBS_DmPD_RotationMove.DigitalOutputControl_01;

{attribute 'TcRpcEnable' := '1'}
METHOD Abort : HRESULT
VAR_INPUT
	hdl : UDINT; // Do not change, used by server.
END_VAR
callCounterAbort := callCounterAbort + 1;
END_METHOD

{attribute 'TcRpcEnable' := '1'}
METHOD CheckState : HRESULT
VAR_INPUT
	hdl : UDINT; // Do not change, used by server.
END_VAR
VAR_OUTPUT
	bBusy : BOOL; // Do not change. Used by server to find out if the job is finished
	
	// List of OutputArguments for OPC UA method, may be customized
	State : BOOL; // Abgeschlossener MethodCall
	MethodCall: BOOL; //Input Recall
END_VAR
callCounterCheckState := callCounterCheckState + 1;
IF NOT jobFinished THEN
	bBusy := TRUE; // job is not finished yet
	CheckState := 0; // no error
ELSE
	bBusy := FALSE; // job is finished
	CheckState := 0; // done, no error occured during execution (OPC UA StatusCode "GOOD")
	jobFinished := FALSE;
	State := ResetMethodCall;
	MethodCall := MethodCall_RotationMove;
END_IF
END_METHOD

{attribute 'TcRpcEnable' := '1'}
METHOD Start : HRESULT
VAR_INPUT
	// List of InputArguments for OPC UA method, may be customized
	MethodCall : BOOL; // some description
	DirectionPoint : STRING;		
END_VAR
VAR_OUTPUT
	hdl : UDINT; // Do not change, used by server.
END_VAR
callCounterStart := callCounterStart + 1;

MethodCall_RotationMove := MethodCall;
DirectionRotation := DirectionPoint;

jobRunning := TRUE;
Start := 0; // no error occured, e.g. while parsing the input arguments (0 = OPC UA StatusCode "GOOD")
END_METHOD

END_FUNCTION_BLOCK

// ---- POUs/Moduls/MBS_Skills/MBS_DmPD_AS_HorizontalMove.TcPOU
{attribute 'OPC.UA.DA.JobMethod' := 'JobMethode_CompressorControl'}
FUNCTION_BLOCK MBS_DmPD_AS_HorizontalMove
VAR
	AlwaysTrue : BOOL := TRUE;
	// Used for debugging purposes to display InputArguments of method call
	MethodCall_CompressorControl : BOOL := FALSE; // used to store InputArg "MethodCall" from Start() method
	ResetMethodCall	: BOOL := FALSE;
	DestinationVertical : STRING;
	PowerOFF_SelfSet : BOOL;
	PowerOFFDelay_SelfSet : TIME;
	callCounterStart : ULINT; // counts how many times the Start() method has been called
	callCounterCheckState : ULINT; // counts how many times the CheckState() method has been called
	callCounterAbort : ULINT; // counts how many times the Abort() method has been called
	
	// Variables to determine if a job has been started (Start() method has been called) or finished
	jobRunning : BOOL;
	jobFinished : BOOL;

	// State machine variable
	state : UDINT;
	
	//Variablen des Transport FBs
	MBS_DmPD_VerticalMove : CompressorControl;
END_VAR
	
VAR_INPUT
	ESS: BOOL;
	TouchSensor_01 : BOOL;
	TON_PowerOnDelay_Compressor : TIME;
	TON_PowerOnDelay_Valve : TIME;
	AutomaticMode: BOOL;
END_VAR

VAR_OUTPUT
	DO_ControlCompressorDmPD_01 : BOOL;
	DO_ControlValveDmPD_02 : BOOL;
END_VAR

MBS_DmPD_VerticalMove(
    MethodCall := MethodCall_CompressorControl,
    EmergencyStopSignal := ESS,
    Destination := DestinationVertical,
    InitStateDrive_Input := ,
    DI01 := TouchSensor_01,
    DI02 := ,
    DI03_EncoderStart01 := ,
    DI04_EncoderStart02 := ,
    DI05_EncoderStart03 := ,
    DI06_EncoderStart04 := ,
    DI07_EncoderStart05 := ,
    DI08_EncoderStart06 := ,
    DI09_EncoderTarget01 := ,
    DI10_EncoderTarget02 := ,
    DI11_EncoderTarget03 := ,
    DI12_EncoderTarget04 := ,
    DI13_EncoderTarget05 := ,
    DI14_EncoderTarget06 := ,
    PowerOFF_SelfSet := PowerOFF_SelfSet,
    TON_Time_PowerOFFSelfSet := PowerOFFDelay_SelfSet,
    TON_Time_Compressor := TON_PowerOnDelay_Compressor,
    TON_Time_Valve := TON_PowerOnDelay_Valve,
    OperatingMode := AutomaticMode
);
DO_ControlCompressorDmPD_01 := MBS_DmPD_VerticalMove.DigitalOutputControl_01;

{attribute 'TcRpcEnable' := '1'}
METHOD Abort : HRESULT
VAR_INPUT
	hdl : UDINT; // Do not change, used by server.
END_VAR
callCounterAbort := callCounterAbort + 1;
END_METHOD

{attribute 'TcRpcEnable' := '1'}
METHOD CheckState : HRESULT
VAR_INPUT
	hdl : UDINT; // Do not change, used by server.
END_VAR
VAR_OUTPUT
	bBusy : BOOL; // Do not change. Used by server to find out if the job is finished
	
	// List of OutputArguments for OPC UA method, may be customized
	State : BOOL; // Abgeschlossener MethodCall
	MethodCall: BOOL; //Input Recall
END_VAR
callCounterCheckState := callCounterCheckState + 1;
IF NOT jobFinished THEN
	bBusy := TRUE; // job is not finished yet
	CheckState := 0; // no error
ELSE
	bBusy := FALSE; // job is finished
	CheckState := 0; // done, no error occured during execution (OPC UA StatusCode "GOOD")
	jobFinished := FALSE;
	State := ResetMethodCall;
	MethodCall := MethodCall_CompressorControl;
END_IF
END_METHOD

{attribute 'TcRpcEnable' := '1'}
METHOD Start : HRESULT
VAR_INPUT
	// List of InputArguments for OPC UA method, may be customized
	MethodCall : BOOL; // some description
	DestinationPoint : STRING;
	SelfSetPowerOff : BOOL;
	SelfSetPowerOffDelay : TIME;	
END_VAR
VAR_OUTPUT
	hdl : UDINT; // Do not change, used by server.
END_VAR
callCounterStart := callCounterStart + 1;

MethodCall_CompressorControl := MethodCall;
DestinationVertical := DestinationPoint;
PowerOFF_SelfSet := SelfSetPowerOff;
PowerOFFDelay_SelfSet := SelfSetPowerOffDelay;

jobRunning := TRUE;
Start := 0; // no error occured, e.g. while parsing the input arguments (0 = OPC UA StatusCode "GOOD")
END_METHOD

END_FUNCTION_BLOCK

// ---- POUs/Moduls/MBS_Skills/MBS_MR02_AS_CuttingProcess.TcPOU
{attribute 'OPC.UA.DA.JobMethod' := 'JobMethode_CuttingProcess'}
FUNCTION_BLOCK MBS_MR02_AS_CuttingProcess
VAR
	AlwaysTrue : BOOL := TRUE;
	// Used for debugging purposes to display InputArguments of method call
	MethodCall_CuttingProcess : BOOL := FALSE; // used to store InputArg "MethodCall" from Start() method
	ResetMethodCall	: BOOL := FALSE;
	ProcessingTime_CuttingProcess : TIME;
	callCounterStart : ULINT; // counts how many times the Start() method has been called
	callCounterCheckState : ULINT; // counts how many times the CheckState() method has been called
	callCounterAbort : ULINT; // counts how many times the Abort() method has been called
	
	// Variables to determine if a job has been started (Start() method has been called) or finished
	jobRunning : BOOL;
	jobFinished : BOOL;

	// State machine variable
	state : UDINT;
	
	//Variablen des FBs
	MBS_MR02_CuttingProcess : CuttingProcess;
END_VAR
	
VAR_INPUT
	ESS: BOOL;
	TouchSensor_01 : BOOL;
	AutomaticMode : BOOL;
END_VAR

VAR_OUTPUT
	DO_CuttingProcessControlMR02 : BOOL;
END_VAR

MBS_MR02_CuttingProcess(
    MethodCall := MethodCall_CuttingProcess,
    EmergencyStopSignal := ESS,
    InitStateDrive_Input := ,
    DI01 := TouchSensor_01,
    TOF_Time_CuttingTime := ProcessingTime_CuttingProcess,
    OperatingMode := AutomaticMode
);
DO_CuttingProcessControlMR02 := MBS_MR02_CuttingProcess.DigitalOutputControl_01;

{attribute 'TcRpcEnable' := '1'}
METHOD Abort : HRESULT
VAR_INPUT
	hdl : UDINT; // Do not change, used by server.
END_VAR
callCounterAbort := callCounterAbort + 1;
END_METHOD

{attribute 'TcRpcEnable' := '1'}
METHOD CheckState : HRESULT
VAR_INPUT
	hdl : UDINT; // Do not change, used by server.
END_VAR
VAR_OUTPUT
	bBusy : BOOL; // Do not change. Used by server to find out if the job is finished
	
	// List of OutputArguments for OPC UA method, may be customized
	State : BOOL; // Abgeschlossener MethodCall
	MethodCall: BOOL; //Input Recall
END_VAR
callCounterCheckState := callCounterCheckState + 1;
IF NOT jobFinished THEN
	bBusy := TRUE; // job is not finished yet
	CheckState := 0; // no error
ELSE
	bBusy := FALSE; // job is finished
	CheckState := 0; // done, no error occured during execution (OPC UA StatusCode "GOOD")
	jobFinished := FALSE;
	State := ResetMethodCall;
	MethodCall := MethodCall_CuttingProcess;
END_IF
END_METHOD

{attribute 'TcRpcEnable' := '1'}
METHOD Start : HRESULT
VAR_INPUT
	// List of InputArguments for OPC UA method, may be customized
	MethodCall : BOOL; // some description
	ProcessingTime : TIME;
END_VAR
VAR_OUTPUT
	hdl : UDINT; // Do not change, used by server.
END_VAR
callCounterStart := callCounterStart + 1;

MethodCall_CuttingProcess := MethodCall;
ProcessingTime_CuttingProcess := ProcessingTime;

jobRunning := TRUE;
Start := 0; // no error occured, e.g. while parsing the input arguments (0 = OPC UA StatusCode "GOOD")
END_METHOD

END_FUNCTION_BLOCK

// ---- POUs/Moduls/MBS_Skills/MBS_CB_AS_HorizontalMove.TcPOU
{attribute 'OPC.UA.DA.JobMethod' := 'JobMethode_HorizontalMove'}
FUNCTION_BLOCK MBS_CB_AS_HorizontalMove
VAR
	AlwaysTrue : BOOL := TRUE;
	// Used for debugging purposes to display InputArguments of method call
	MethodCall_HorizontalMove : BOOL := FALSE; // used to store InputArg "MethodCall" from Start() method
	ResetMethodCall	: BOOL := FALSE;	
	DirectionHorizontal : STRING; // defines movement direction
	callCounterStart : ULINT; // counts how many times the Start() method has been called
	callCounterCheckState : ULINT; // counts how many times the CheckState() method has been called
	callCounterAbort : ULINT; // counts how many times the Abort() method has been called
	
	// Variables to determine if a job has been started (Start() method has been called) or finished
	jobRunning : BOOL;
	jobFinished : BOOL;

	// State machine variable
	state : UDINT;
	
	// FB Intatziation Variable
	MBS_CB_HorizontalMove : AxisControl_MultipleInputSensors;
END_VAR
	
VAR_INPUT
	ESS: BOOL;
	TouchSensor_01 : BOOL;
	LightSensor_01 : BOOL;
	TOF_Time_MotorControl : TIME;
	AutomaticMode: BOOL;
END_VAR

VAR_OUTPUT
	DO_MovingHorizontalCB_01 : BOOL;
END_VAR

MBS_CB_HorizontalMove(
    MethodCall := MethodCall_HorizontalMove,
    EmergencyStopSignal := ESS,
    Direction := DirectionHorizontal,
    InitStateDrive_Input := ,
    DI01 := TouchSensor_01,
    DI02 := LightSensor_01,
    TouchSensorRelief := ,
    TOF_Time_MotorControl := TOF_Time_MotorControl,
    TOF_Time_TouchSensorRelief := ,
    OperatingMode := AutomaticMode
);
DO_MovingHorizontalCB_01 := MBS_CB_HorizontalMove.DigitalOutputControl_01;

{attribute 'TcRpcEnable' := '1'}
METHOD Abort : HRESULT
VAR_INPUT
	hdl : UDINT; // Do not change, used by server.
END_VAR
callCounterAbort := callCounterAbort + 1;
END_METHOD

{attribute 'TcRpcEnable' := '1'}
METHOD CheckState : HRESULT
VAR_INPUT
	hdl : UDINT; // Do not change, used by server.
END_VAR
VAR_OUTPUT
	bBusy : BOOL; // Do not change. Used by server to find out if the job is finished
	
	// List of OutputArguments for OPC UA method, may be customized
	State : BOOL; // Abgeschlossener MethodCall
	MethodCall: BOOL; //Input Recall
END_VAR
callCounterCheckState := callCounterCheckState + 1;
IF NOT jobFinished THEN
	bBusy := TRUE; // job is not finished yet
	CheckState := 0; // no error
ELSE
	bBusy := FALSE; // job is finished
	CheckState := 0; // done, no error occured during execution (OPC UA StatusCode "GOOD")
	jobFinished := FALSE;
	State := ResetMethodCall;
	MethodCall := MethodCall_HorizontalMove;
END_IF
END_METHOD

{attribute 'TcRpcEnable' := '1'}
METHOD Start : HRESULT
VAR_INPUT
	// List of InputArguments for OPC UA method, may be customized
	MethodCall : BOOL; // some description
	DirectionPoint : STRING;	
END_VAR
VAR_OUTPUT
	hdl : UDINT; // Do not change, used by server.
END_VAR
callCounterStart := callCounterStart + 1;

MethodCall_HorizontalMove := MethodCall;
DirectionHorizontal := DirectionPoint;

jobRunning := TRUE;
Start := 0; // no error occured, e.g. while parsing the input arguments (0 = OPC UA StatusCode "GOOD")
END_METHOD

END_FUNCTION_BLOCK

